// TIA Portal project "项目1_V15.1" (V15.1)

(* hardware
DEVICE "S7-1200 station_2"  S7-1200 Station
   slot 0: "Rack_0"  S7-1200 Rack  Rack  V1.0
   slot 1: "300-1PLC"  CPU 1214C DC/DC/DC  6ES7 214-1AG40-0XB0  V4.2
   slot 2: "DI 16/DQ 16x24VDC_1"  6ES7 223-1BL32-0XB0  V2.0
   slot 3: "DI 16/DQ 16x24VDC_2"  6ES7 223-1BL32-0XB0  V2.0
   slot 4: "DI 8x24VDC_1"  6ES7 221-1BF32-0XB0  V2.0
   slot 5: "AI 4x13BIT/AQ 2x14BIT_1"  6ES7 234-4HE32-0XB0  V2.0
DEVICE "GSD device_9"  GSD.Device.PN
   slot 0: "机架"  Rack  V1.0
   slot 0: "输入轴伺服"  SINAMICS V90 PN V1.0  6SL3 210-5Fxxx-xxFx  V1.00
      slot 0: "SINAMICS V90 PN V1.0"  SINAMICS V90 PN V1.0
      slot 1: "PN-IO"  PN-IO
         slot 1: "端口1"  Port 1
         slot 2: "端口2"  Port 2
      slot 1: "驱动_1"  Drive
         slot 0: "模块访问点"  Module Access Point
         slot 1: "没有 PROFIsafe"  without PROFIsafe
   slot 2: "标准报文3, PZD-5/9"  Standard telegram 3, PZD-5/9
DEVICE "GSD device_8"  GSD.Device.PN
   slot 0: "机架"  Rack  V1.0
   slot 0: "输入轴移载"  SINAMICS V90 PN V1.0  6SL3 210-5Fxxx-xxFx  V1.00
      slot 0: "SINAMICS V90 PN V1.0"  SINAMICS V90 PN V1.0
      slot 1: "PN-IO"  PN-IO
         slot 1: "端口1"  Port 1
         slot 2: "端口2"  Port 2
      slot 1: "驱动_1"  Drive
         slot 0: "模块访问点"  Module Access Point
         slot 1: "没有 PROFIsafe"  without PROFIsafe
   slot 2: "标准报文3, PZD-5/9"  Standard telegram 3, PZD-5/9
DEVICE "GSD device_10"  GSD.Device.PN
   slot 0: "机架"  Rack  V1.0
   slot 0: "工装移载"  SINAMICS V90 PN V1.0  6SL3 210-5Fxxx-xxFx  V1.00
      slot 0: "SINAMICS V90 PN V1.0"  SINAMICS V90 PN V1.0
      slot 1: "PN-IO"  PN-IO
         slot 1: "端口1"  Port 1
         slot 2: "端口2"  Port 2
      slot 1: "驱动_1"  Drive
         slot 0: "模块访问点"  Module Access Point
         slot 1: "没有 PROFIsafe"  without PROFIsafe
   slot 2: "标准报文3, PZD-5/9"  Standard telegram 3, PZD-5/9
*)

// ===== PLC "300-1PLC"  CPU 1214C DC/DC/DC =====

VAR_GLOBAL   // PLC tag table "默认变量表"
   "角度编码器A" AT %I0.0 : Bool;
   "角度编码器B" AT %I0.1 : Bool;
   "角度编码器Z" AT %I0.2 : Bool;
   "在位传感器" AT %I1.4 : Bool;
   "输入轴扶持气缸进到位" AT %I2.0 : Bool;
   "输入轴扶持气缸退到位" AT %I2.1 : Bool;
   "产品夹紧气缸1进到位" AT %I2.2 : Bool;
   "产品夹紧气缸1退到位" AT %I2.3 : Bool;
   "产品夹紧气缸2进到位" AT %I2.5 : Bool;
   "产品夹紧气缸2退到位" AT %I2.4 : Bool;
   "产品定位气缸进到位" AT %I2.6 : Bool;
   "产品定位气缸退到位" AT %I2.7 : Bool;
   "振动检测气缸1进到位" AT %I3.0 : Bool;
   "振动检测气缸1退到位" AT %I3.1 : Bool;
   "振动检测气缸2进到位" AT %I3.2 : Bool;
   "振动检测气缸2退到位" AT %I3.3 : Bool;
   "输出轴花键移载气缸进到位" AT %I3.4 : Bool;
   "输出轴花键移载气缸退到位" AT %I3.5 : Bool;
   "安全门气缸进到位" AT %I3.6 : Bool;
   "安全门气缸退到位" AT %I3.7 : Bool;
   "启动" AT %I4.0 : Bool;
   "复位" AT %I4.1 : Bool;
   "手自动" AT %I4.2 : Bool;
   "安全继电器急停" AT %I4.3 : Bool;
   "安全门开关" AT %I4.4 : Bool;
   "急停" AT %I4.5 : Bool;
   "报警1" AT %I5.0 : Bool;
   "报警2" AT %I5.1 : Bool;
   "报警3" AT %I5.2 : Bool;
   "报警4" AT %I5.3 : Bool;
   "扭矩传感器1" AT %IW144 : Int;
   "扭矩传感器2-1" AT %IW146 : Int;
   "扭矩传感器2-2" AT %IW148 : Int;
   "电流传感器" AT %IW150 : Int;
   "输入轴移载伺服_LowHwLimitSwitch" AT %I0.4 : Bool;
   "输入轴移载伺服_HighHwLimitSwitch" AT %I0.3 : Bool;
   "输入轴移载伺服_归位开关" AT %I0.5 : Bool;
   "工装移载伺服_Drive_IN" AT %I104.0 : "PD_TEL3_IN";
   "工装移载伺服_LowHwLimitSwitch" AT %I0.7 : Bool;
   "工装移载伺服_HighHwLimitSwitch" AT %I0.6 : Bool;
   "工装移载伺服_归位开关" AT %I1.0 : Bool;
   "角度编码器" AT %ID1000 : DInt;
   "气源不足指示" AT %I5.4 : Bool;
   "安全光栅" AT %I4.7 : Bool;
   "工件在位" AT %I1.1 : Bool;
   "输入轴驱动伺服_Drive_IN" AT %I68.0 : "PD_TEL1_IN";
   "输入轴移载伺服_Drive_IN" AT %I86.0 : "PD_TEL3_IN";
   "输入轴驱动伺服_Encoder_IN" AT %I68.0 : "PD_TEL3_IN";
   "复位1" AT %Q0.0 : Bool;
   "复位2" AT %Q0.1 : Bool;
   "复位3" AT %Q0.2 : Bool;
   "复位4" AT %Q0.3 : Bool;
   "点火" AT %Q0.4 : Bool;
   "转速" AT %Q0.5 : Bool;
   "车速" AT %Q0.6 : Bool;
   "输入轴扶持气缸进" AT %Q2.0 : Bool;
   "输入轴扶持气缸退" AT %Q2.1 : Bool;
   "产品松开" AT %Q2.2 : Bool;
   "产品夹紧" AT %Q2.3 : Bool;
   "支架松开" AT %Q2.4 : Bool;
   "支架夹紧" AT %Q2.5 : Bool;
   "产品定位气缸进" AT %Q3.6 : Bool;
   "产品定位气缸退" AT %Q3.7 : Bool;
   "振动检测气缸1进" AT %Q3.0 : Bool;
   "振动检测气缸1退" AT %Q3.1 : Bool;
   "振动检测气缸2进" AT %Q3.2 : Bool;
   "振动检测气缸2退" AT %Q3.3 : Bool;
   "输出轴花键移载气缸进" AT %Q2.6 : Bool;
   "输出轴花键移载气缸退" AT %Q2.7 : Bool;
   "安全门气缸进" AT %Q3.4 : Bool;
   "安全门气缸退" AT %Q3.5 : Bool;
   "三色灯-红" AT %Q4.0 : Bool;
   "三色灯-黄" AT %Q4.1 : Bool;
   "三色灯-绿" AT %Q4.2 : Bool;
   "蜂鸣器" AT %Q4.3 : Bool;
   "两色灯-红" AT %Q4.4 : Bool;
   "两色灯-绿" AT %Q4.5 : Bool;
   "总气阀" AT %Q4.6 : Bool;
   "工位复位中" AT %Q4.7 : Bool;
   "30V电源控制" AT %QW144 : Int;
   "输入轴移载伺服_Drive_OUT" AT %Q74.0 : "PD_TEL3_OUT";
   "工装移载伺服_Drive_OUT" AT %Q84.0 : "PD_TEL3_OUT";
   "输入轴旋转-已复位" AT %Q6.0 : Bool;
   "输入轴移载-已复位" AT %Q6.1 : Bool;
   "工装移载-已复位" AT %Q6.2 : Bool;
   "T1T2切换" AT %Q5.0 : Bool;
   "输入轴驱动伺服_Drive_OUT" AT %Q64.0 : "PD_TEL3_OUT";
   "System_Byte" AT %MB1 : Byte;
   "FirstScan" AT %M1.0 : Bool;
   "DiagStatusUpdate" AT %M1.1 : Bool;
   "AlwaysTRUE" AT %M1.2 : Bool;
   "AlwaysFALSE" AT %M1.3 : Bool;
   "Clock_Byte" AT %MB0 : Byte;
   "Clock_10Hz" AT %M0.0 : Bool;
   "Clock_5Hz" AT %M0.1 : Bool;
   "Clock_2.5Hz" AT %M0.2 : Bool;
   "Clock_2Hz" AT %M0.3 : Bool;
   "Clock_1.25Hz" AT %M0.4 : Bool;
   "Clock_1Hz" AT %M0.5 : Bool;
   "Clock_0.625Hz" AT %M0.6 : Bool;
   "Clock_0.5Hz" AT %M0.7 : Bool;
   "Car_speed" AT %MD2000 : Real;
   "Engine_Speed" AT %MD2004 : Real;
   "复位启动" AT %M100.0 : Bool;
   "复位完成" AT %M100.1 : Bool;
   "程序停止" AT %M100.2 : Bool;
   "电机控制器启动" AT %M99.0 : Bool;
   "电机正转启动" AT %M99.1 : Bool;
   "电机反转启动" AT %M99.2 : Bool;
   "Tag_1" AT %MW1000 : Word;
   "Tag_2" AT %MW1024 : Word;
   "Tag_3" AT %MW1345 : Word;
   "Tag_4" AT %MW1456 : Word;
   "转速方向" AT %Q0.7 : Bool;
   "车速方向" AT %Q1.0 : Bool;
END_VAR

TYPE "In_config"
VERSION : 0.1
   STRUCT
      接近位移 : Real;
      接近速度 : Real;
      套入位移 : Real;
      套入速度 : Real;
      摆动参数 : "In_swing_config";
   END_STRUCT;
END_TYPE

TYPE "In_swing_config"
VERSION : 0.1
   STRUCT
      启用状态 : Real;
      摆动速度 : Real;
      摆动角度 : Real;
      保护扭矩 : Real;
   END_STRUCT;
END_TYPE

TYPE "Fixture_transfer_config"
VERSION : 0.1
   STRUCT
      定位位置 : Real;
      定位速度 : Real;
   END_STRUCT;
END_TYPE

TYPE "Test_No_Load_CFG"
VERSION : 0.1
   STRUCT
      启用助力 : Real := 0.0;
      空载速度 : Real := 0.0;
      空载位移 : Real := 0.0;
      扭矩保护 : Real := 0.0;
   END_STRUCT;
END_TYPE

TYPE "Test_Function_CFG"
VERSION : 0.1
   STRUCT
      试验速度 : Real;
      试验角度 : Real;
      负载扭矩 : Real;
      保护扭矩 : Real;
   END_STRUCT;
END_TYPE

TYPE "Test_Input&Output_Characteristics_CFG"
VERSION : 0.1
   STRUCT
      试验速度 : Real;
      换向扭矩 : Real;
      模拟车速 : Real;
      模拟发动机转速 : Real;
   END_STRUCT;
END_TYPE

TYPE "Test_NVH"
VERSION : 0.1
   STRUCT
      检测点1 : Real;
      检测点2 : Real;
      正向检测时间 : Real;
      逆向检测时间 : Real;
   END_STRUCT;
END_TYPE

DATA_BLOCK "MB_TCON_Rapid"   // DB5
{ S7_Optimized_Access := 'TRUE' }
VERSION : 0.1
   VAR
      MB_SERVER : TCON_IP_v4;
   END_VAR
BEGIN
   MB_SERVER.InterfaceId := 64;
   MB_SERVER.ID := 1;
   MB_SERVER.LocalPort := 502;
END_DATA_BLOCK

DATA_BLOCK "Modbus_Data_Rapid"   // DB6
{ S7_Optimized_Access := 'FALSE' }
VERSION : 0.1
   VAR
      设备编号 : Int := 0;
      产品型号 : Int := 0;
      设备状态 : Int;
      错误代码 : Int;
      当前曲线 : Int;
      传感器标定值 : Array[0..7] of Real;
   END_VAR
BEGIN
   // 传感器标定值[0] : 输入轴驱动伺服位移
   // 传感器标定值[1] : 输入轴移载伺服位移
   // 传感器标定值[2] : 工装移载伺服位移
   // 传感器标定值[3] : 输入轴编码器
   // 传感器标定值[4] : 输入轴扭矩
   // 传感器标定值[5] : 输出轴扭矩小量程
   // 传感器标定值[6] : 输出轴扭矩大量程
   // 传感器标定值[7] : 吸收电流
END_DATA_BLOCK

DATA_BLOCK "Modbus_Data"   // DB7
{ S7_Optimized_Access := 'FALSE' }
VERSION : 0.1
   VAR
      输入扭矩传感器参数 : Array[0..1] of Real;   // AF400001L2
      输出扭矩传感器参数小量程 : Array[0..1] of Real;   // AF400005L2
      输出扭矩传感器参数大量程 : Array[0..1] of Real;   // AF400009L2
      电流传感器参数 : Array[0..1] of Real;   // AF400013L2
      输入轴自动参数 : "In_config";   // AF400017L4
      输入轴移载手动参数 : Array[0..3] of Real;   // AF400025L4
      输入轴旋转参数 : Array[0..3] of Real;   // AF400041L4
      工装移载参数 : "Fixture_transfer_config";   // AF400049L4
      工装移载手动参数 : Array[0..3] of Real;   // AF400057L4
      空载试验参数 : "Test_No_Load_CFG";   // AF400065L4
      功能试验参数 : "Test_Function_CFG";   // AF400073L4
      力特性试验参数 : "Test_Input&Output_Characteristics_CFG";   // AF400081L4
      逆向空载试验参数 : "Test_No_Load_CFG";   // AF400097L4
      振动NVH试验参数 : "Test_NVH";   // AF400097L4
   END_VAR
BEGIN
   输出扭矩传感器参数小量程[0] := 0.0;   // 量程下限
   输出扭矩传感器参数小量程[1] := 20.0;   // 量程上限
   输出扭矩传感器参数大量程[1] := 233.0;   // 量程上限（校验值233）
   输出扭矩传感器参数大量程[0] := 0.0;   // 量程下限
   输入扭矩传感器参数[1] := 58.0;   // 量程上限(校验值48.0)
   输入扭矩传感器参数[0] := 0.0;   // 量程下限
   电流传感器参数[0] := -100.0;   // 量程下限
   电流传感器参数[1] := 100.0;   // 量程下限
   // 输入轴移载手动参数[0] : 手动状态
   // 输入轴移载手动参数[1] : 手动速度
   // 输入轴移载手动参数[2] : 相对定位
   // 输入轴移载手动参数[3] : 绝对定位
   // 输入轴旋转参数[0] : 手动状态
   // 输入轴旋转参数[1] : 手动速度
   // 输入轴旋转参数[2] : 相对定位
   // 输入轴旋转参数[3] : 绝对定位
   // 工装移载手动参数[0] : 手动状态
   // 工装移载手动参数[1] : 手动速度
   // 工装移载手动参数[2] : 相对定位
   // 工装移载手动参数[3] : 绝对定位
END_DATA_BLOCK

DATA_BLOCK "MB_TCON"   // DB9
{ S7_Optimized_Access := 'TRUE' }
VERSION : 0.1
   VAR
      MB_SERVER : TCON_IP_v4;
   END_VAR
BEGIN
   MB_SERVER.InterfaceId := 64;
   MB_SERVER.ID := 2;
   MB_SERVER.LocalPort := 502;
END_DATA_BLOCK

DATA_BLOCK "Reset_DB"   // DB11
{ S7_Optimized_Access := 'TRUE' }
VERSION : 0.1
// stored: InstanceOfName Reset
"Reset"
BEGIN
END_DATA_BLOCK

DATA_BLOCK "Alarm_DB"   // DB15
{ S7_Optimized_Access := 'TRUE' }
VERSION : 0.1
// stored: InstanceOfName Alarm
"Alarm"
BEGIN
END_DATA_BLOCK

DATA_BLOCK "All_Servo_DB"   // DB18
{ S7_Optimized_Access := 'TRUE' }
VERSION : 0.1
// stored: InstanceOfName All_Servo
"All_Servo"
BEGIN
END_DATA_BLOCK

DATA_BLOCK "设置电压_DB"   // DB20
{ S7_Optimized_Access := 'TRUE' }
VERSION : 0.1
// stored: InstanceOfName 设置电压
"设置电压"
BEGIN
END_DATA_BLOCK

DATA_BLOCK "Auto_DB"   // DB21
{ S7_Optimized_Access := 'TRUE' }
VERSION : 0.1
// stored: InstanceOfName Auto
"Auto"
BEGIN
END_DATA_BLOCK

DATA_BLOCK "左右摆动_DB"   // DB22
{ S7_Optimized_Access := 'TRUE' }
VERSION : 0.1
// stored: InstanceOfName 左右摆动
"左右摆动"
BEGIN
END_DATA_BLOCK

// folder: System blocks/Program resources

DATA_BLOCK "IEC_Timer_0_DB"   // DB19
{ S7_Optimized_Access := 'TRUE' }
AUTHOR : Simatic
FAMILY : IEC
NAME : IEC_TMR
VERSION : 1.0
// stored: InstanceOfName IEC_TIMER
"IEC_TIMER"
BEGIN
END_DATA_BLOCK

// folder: (top level)

DATA_BLOCK "输入轴驱动伺服"   // DB1, Motion_DB
{ S7_Optimized_Access := 'TRUE' }
AUTHOR : SIMATIC
FAMILY : BasicMC
NAME : TO_PosAx
VERSION : 6.0
// stored: InstanceOfName TO_PositioningAxis
"TO_PositioningAxis"
BEGIN
   // Axis.Encoder.TelegramAddressOutCU = %Q64.0
   // Axis.Encoder.TelegramAddressInCU = %I68.0
   // Axis.Encoder.DoNameCU = 输入轴伺服.驱动_1_编码器1
   // Axis.Drive.OutputAddress = 64
   // Axis.Drive.InputAddress = 68
   // Axis.Encoder.OutputAddress = 64
   // Axis.Encoder.InputAddress = 68
   // Axis.Drive.TelegramAddressOutCU = %Q64.0
   // Axis.Drive.TelegramAddressInCU = %I68.0
   // Axis.Drive.TelegramType = 2
   // Axis.Drive.DoNameCU = 输入轴伺服.驱动_1
   // Axis.LengthUnit.LastDistance = 1005
   // Axis.LengthUnitNormalized.Distance = 1005
   // Axis.Encoder.SelectedHscIndexCU = -1
   // Axis.Encoder.DbTypeCU = Classic
   // Axis.Drive.DbTypeCU = Classic
END_DATA_BLOCK

DATA_BLOCK "输入轴移载伺服"   // DB2, Motion_DB
{ S7_Optimized_Access := 'TRUE' }
AUTHOR : SIMATIC
FAMILY : BasicMC
NAME : TO_PosAx
VERSION : 6.0
// stored: InstanceOfName TO_PositioningAxis
"TO_PositioningAxis"
BEGIN
   // Axis.Encoder.TelegramAddressOutCU = %Q74.0
   // Axis.Encoder.TelegramAddressInCU = %I86.0
   // Axis.Encoder.DoNameCU = 输入轴移载.驱动_1_编码器1
   // Axis.Drive.OutputAddress = 74
   // Axis.Drive.InputAddress = 86
   // Axis.Encoder.OutputAddress = 74
   // Axis.Encoder.InputAddress = 86
   // Axis.Drive.TelegramAddressOutCU = %Q74.0
   // Axis.Drive.TelegramAddressInCU = %I86.0
   // Axis.Drive.TelegramType = 2
   // Axis.Drive.DoNameCU = 输入轴移载.驱动_1
   // Axis.HomingReferencePointSwitch_AddressCU = %I0.5
   // Axis.PositionLimitsMax_AddressCU = %I0.3
   // Axis.PositionLimitsMin_AddressCU = %I0.4
   // Axis.LengthUnitNormalized.Distance = 1013
   // Axis.Encoder.SelectedHscIndexCU = -1
   // Axis.Encoder.DbTypeCU = Classic
   // Axis.Drive.DbTypeCU = Classic
END_DATA_BLOCK

DATA_BLOCK "工装移载伺服"   // DB3, Motion_DB
{ S7_Optimized_Access := 'TRUE' }
AUTHOR : SIMATIC
FAMILY : BasicMC
NAME : TO_PosAx
VERSION : 6.0
// stored: InstanceOfName TO_PositioningAxis
"TO_PositioningAxis"
BEGIN
   // Axis.Encoder.TelegramAddressOutCU = %Q84.0
   // Axis.Encoder.TelegramAddressInCU = %I104.0
   // Axis.Encoder.DoNameCU = 工装移载.驱动_1_编码器1
   // Axis.Drive.OutputAddress = 84
   // Axis.Drive.InputAddress = 104
   // Axis.Encoder.OutputAddress = 84
   // Axis.Encoder.InputAddress = 104
   // Axis.Drive.TelegramAddressOutCU = %Q84.0
   // Axis.Drive.TelegramAddressInCU = %I104.0
   // Axis.Drive.DoNameCU = 工装移载.驱动_1
   // Axis.HomingReferencePointSwitch_AddressCU = %I1.0
   // Axis.PositionLimitsMax_AddressCU = %I0.6
   // Axis.PositionLimitsMin_AddressCU = %I0.7
   // Axis.Drive.TelegramType = 2
   // Axis.LengthUnitNormalized.Distance = 1013
   // Axis.Encoder.SelectedHscIndexCU = -1
   // Axis.Encoder.DbTypeCU = Classic
   // Axis.Drive.DbTypeCU = Classic
END_DATA_BLOCK

DATA_BLOCK "模拟转速"   // DB16, Motion_DB
{ S7_Optimized_Access := 'TRUE' }
AUTHOR : SIMATIC
FAMILY : BasicMC
NAME : TO_PosAx
VERSION : 6.0
// stored: InstanceOfName TO_PositioningAxis
"TO_PositioningAxis"
BEGIN
   // Axis.OnlinePtoIndexCU = 3
   // Axis.SelectedChannel2EnumCU = %Q1.0
   // Axis.LengthUnit.LastDistance = -1
   // Axis.OnlinePtoModeCUEnumValue = PTO（脉冲 A 和方向 B）
   // Axis.OnlinePtoModeCU = 16#0000_0002
   // Axis.SelectedChannel1EnumCU = %Q0.5
   // Pulse.MinDeltaDeltaFrequencyCU = 0.004
   // Pulse.MaxDeltaDeltaFrequencyCU = 1.0E+10
   // Pulse.MinDeltaFrequencyCU = 0.005
   // Pulse.MaxDeltaFrequencyCU = 9.5E+9
   // Pulse.MinFrequencyCU = 1.0
   // Pulse.MaxFrequencyCU = 30000.0
   // Pulse.OutputSourceCU = 16#0000_0000
   // Axis.SelectPTO = 3
END_DATA_BLOCK

DATA_BLOCK "模拟车速"   // DB17, Motion_DB
{ S7_Optimized_Access := 'TRUE' }
AUTHOR : SIMATIC
FAMILY : BasicMC
NAME : TO_PosAx
VERSION : 6.0
// stored: InstanceOfName TO_PositioningAxis
"TO_PositioningAxis"
BEGIN
   // Axis.OnlinePtoIndexCU = 2
   // Axis.OnlinePtoModeCU = 16#0000_0002
   // Axis.SelectedChannel2EnumCU = %Q0.7
   // Axis.SelectedChannel1EnumCU = %Q0.6
   // Pulse.MinDeltaDeltaFrequencyCU = 0.004
   // Pulse.MaxDeltaDeltaFrequencyCU = 1.0E+10
   // Pulse.MinDeltaFrequencyCU = 0.005
   // Pulse.MaxDeltaFrequencyCU = 9.5E+9
   // Pulse.MinFrequencyCU = 1.0
   // Pulse.MaxFrequencyCU = 30000.0
   // Pulse.OutputSourceCU = 16#0000_0000
   // Axis.SelectPTO = 2
   // Axis.OnlinePtoModeCUEnumValue = PTO（脉冲 A 和方向 B）
   // Axis.LengthUnit.LastDistance = -1
END_DATA_BLOCK

FUNCTION_BLOCK "设置电压"   // FB1, LAD
{ S7_Optimized_Access := 'TRUE' }
VERSION : 0.1
   VAR_INPUT
      电压 : Real;
   END_VAR
BEGIN

REGION Network 1
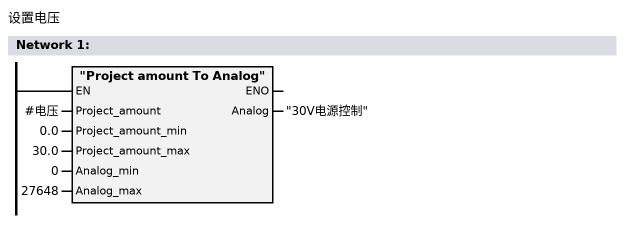
   RUNG wire#powerrail
      "Project amount To Analog"(Project_amount := #电压, Project_amount_min := 0.0, Project_amount_max := 30.0, Analog_min := 0, Analog_max := 27648, Analog => "30V电源控制")
   END_RUNG
   // the same network as SCL:
   "Project amount To Analog"(Project_amount := #电压,
                           Project_amount_min := 0.0,
                           Project_amount_max := 30.0,
                           Analog_min := 0,
                           Analog_max := 27648,
                           Analog => "30V电源控制");
END_REGION
END_FUNCTION_BLOCK

FUNCTION_BLOCK "Servo"   // FB2, LAD
{ S7_Optimized_Access := 'TRUE' }
VERSION : 0.1
   VAR_INPUT
      Axis : TO_PositioningAxis;
      Son : Bool;
      Halt : Bool;
      Stop : Bool;
      Absoulte_Position : Real;
      Relative_Position : Real;
      Velocity : Real;
      JogForword : Bool;
      JogBackword : Bool;
      MoveAbsolute : Bool;
      MoveRelative : Bool;
      MoveHome : Bool;
      Mode : Int;
   END_VAR
   VAR_OUTPUT
      Done : Bool;
   END_VAR
   VAR_IN_OUT
      HomingDone : Bool;
   END_VAR
   VAR
      Temp : Array[0..7] of Bool;
      Reser_Done : Bool;
      MC_Power_Instance : MC_Power;
      MC_Reset_Instance : MC_Reset;
      MC_Home_Instance : MC_Home;
      MC_Halt_Instance : MC_Halt;
      MC_MoveAbsolute_Instance : MC_MoveAbsolute;
      MC_MoveRelative_Instance : MC_MoveRelative;
      MC_MoveJog_Instance : MC_MoveJog;
      IEC_Timer_0_Instance : TP_TIME;
      IEC_Timer_0_Instance_1 : TON_TIME;
      IEC_Timer_0_Instance_2 : TON_TIME;
      MC_ReadParam_Instance : MC_ReadParam;
   END_VAR
   VAR_TEMP   // added for the SCL form of the ladder/FBD networks
      _w1 : Bool;
   END_VAR
BEGIN

REGION Network 1
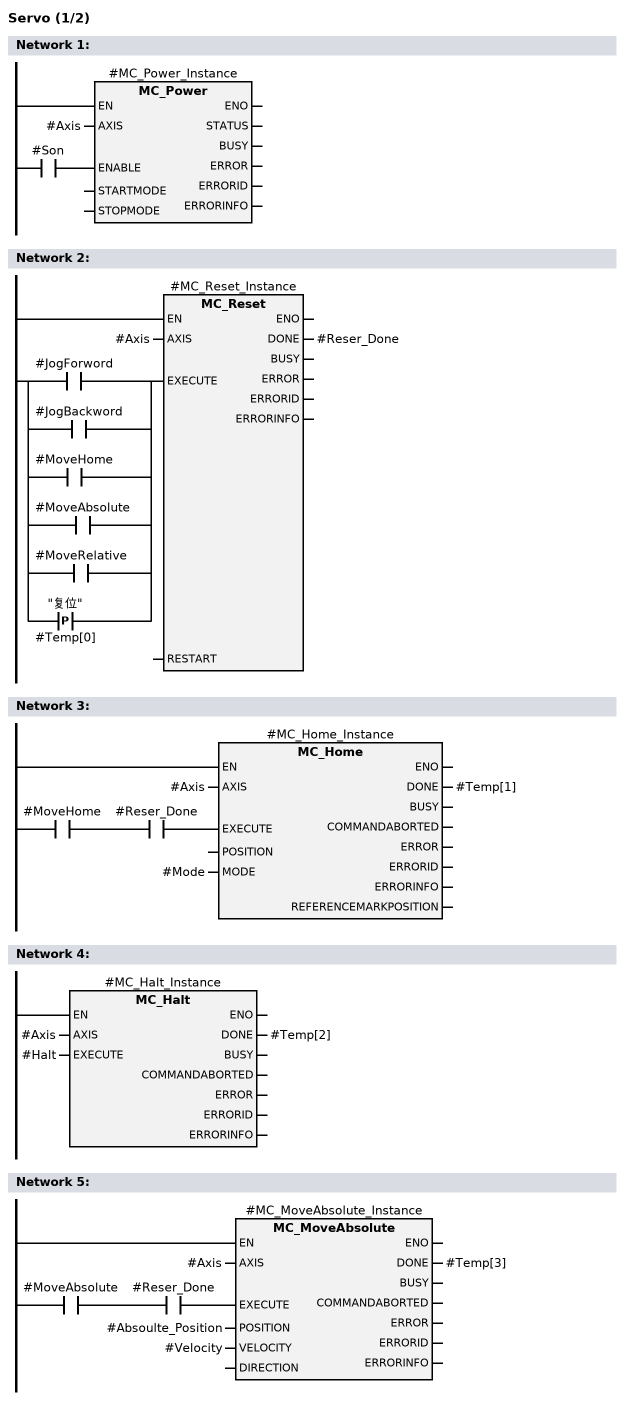
   #MC_Power_Instance(Axis := #Axis, Enable := #Son);   // MC_Power
END_REGION

REGION Network 2
   #_w1 := "复位" AND NOT #Temp[0];   // rising edge of "复位"
   #Temp[0] := "复位";
   #MC_Reset_Instance(Axis := #Axis,   // MC_Reset
                      Execute := #JogForword OR #JogBackword OR #MoveHome OR #MoveAbsolute OR #MoveRelative OR #_w1,
                      Done => #Reser_Done);
END_REGION

REGION Network 3
   #MC_Home_Instance(Axis := #Axis, Execute := #MoveHome AND #Reser_Done, Mode := #Mode, Done => #Temp[1]);   // MC_Home
END_REGION

REGION Network 4
   #MC_Halt_Instance(Axis := #Axis, Execute := #Halt, Done => #Temp[2]);   // MC_Halt
END_REGION

REGION Network 5
   #MC_MoveAbsolute_Instance(Axis := #Axis,   // MC_MoveAbsolute
                           Execute := #MoveAbsolute AND #Reser_Done,
                           Position := #Absoulte_Position,
                           Velocity := #Velocity,
                           Done => #Temp[3]);
END_REGION

REGION Network 6
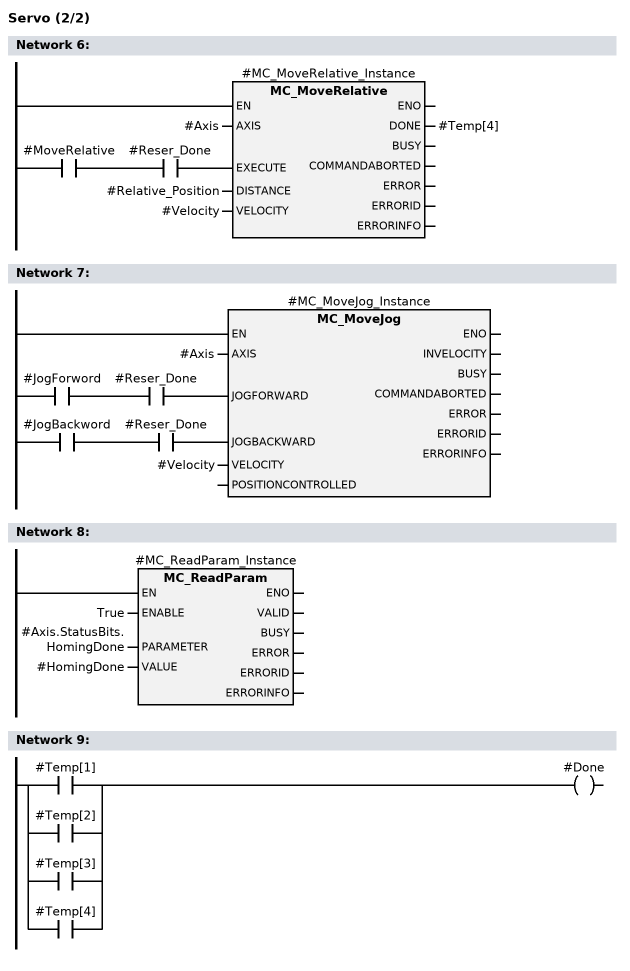
   #MC_MoveRelative_Instance(Axis := #Axis,   // MC_MoveRelative
                           Execute := #MoveRelative AND #Reser_Done,
                           Distance := #Relative_Position,
                           Velocity := #Velocity,
                           Done => #Temp[4]);
END_REGION

REGION Network 7
   #MC_MoveJog_Instance(Axis := #Axis,   // MC_MoveJog
                        JogForward := #JogForword AND #Reser_Done,
                        JogBackward := #JogBackword AND #Reser_Done,
                        Velocity := #Velocity);
END_REGION

REGION Network 8
   #MC_ReadParam_Instance(Enable := True, Parameter := #Axis.StatusBits.HomingDone, Value := #HomingDone);   // MC_ReadParam
END_REGION

REGION Network 9
   RUNG wire#powerrail
      Contact( #Temp[1] )
      wire#w1
      Coil( #Done )
   END_RUNG
   RUNG wire#powerrail
      Contact( #Temp[2] )
   END_RUNG wire#w1
   RUNG wire#powerrail
      Contact( #Temp[3] )
   END_RUNG wire#w1
   RUNG wire#powerrail
      Contact( #Temp[4] )
   END_RUNG wire#w1
   // the same network as SCL:
   #Done := #Temp[1] OR #Temp[2] OR #Temp[3] OR #Temp[4];
END_REGION
END_FUNCTION_BLOCK

FUNCTION_BLOCK "All_Servo"   // FB3, LAD
{ S7_Optimized_Access := 'TRUE' }
VERSION : 0.1
   VAR
      Temp : Array[0..3] of Bool;
      IEC_Timer_0_Instance : TON_TIME;
      IEC_Timer_0_Instance_1 : TP_TIME;
      IEC_Timer_0_Instance_2 : TP_TIME;
      IEC_Timer_0_Instance_3 : TON_TIME;
      IEC_Timer_0_Instance_4 : TP_TIME;
      IEC_Timer_0_Instance_5 : TON_TIME;
      IEC_Timer_0_Instance_6 : TON_TIME;
      Servo_Instance : "Servo";
      Servo_Instance_1 : "Servo";
      Servo_Instance_2 : "Servo";
      Servo_Instance_3 : "Servo";
      MC_Power_Instance : MC_Power;
      MC_Power_Instance_1 : MC_Power;
   END_VAR
   VAR_TEMP   // added for the SCL form of the ladder/FBD networks
      _w1 : Bool;
   END_VAR
BEGIN

REGION Network 1: 输入轴驱动伺服
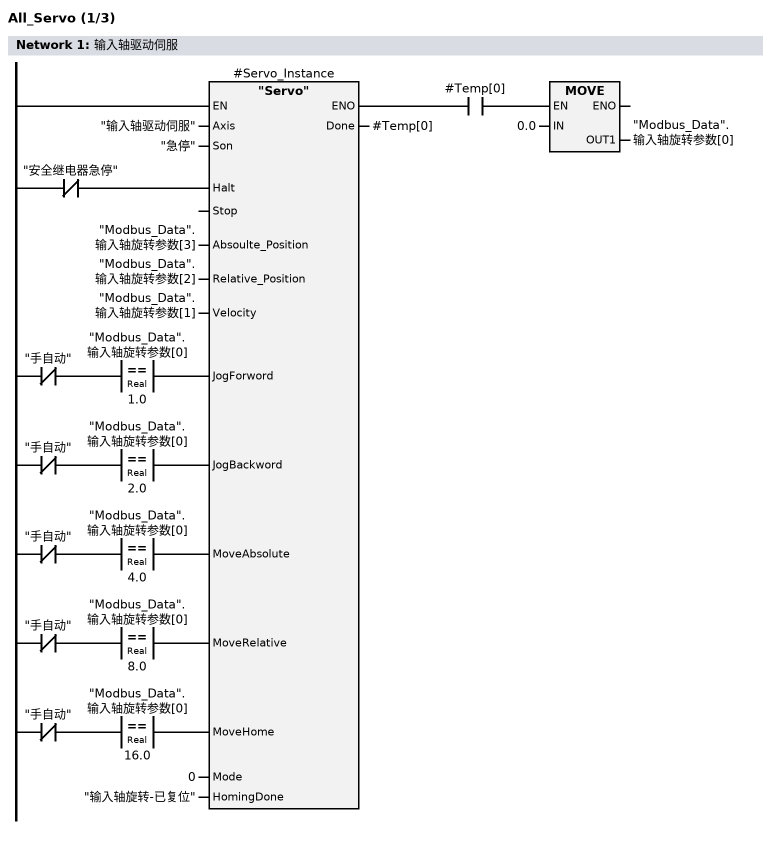
   RUNG wire#powerrail
      #Servo_Instance(Halt := wire#w1, JogForword := wire#w2, JogBackword := wire#w3, MoveAbsolute := wire#w4, MoveRelative := wire#w5, MoveHome := wire#w6, Axis := "输入轴驱动伺服", Son := "急停", Stop :=, Absoulte_Position := "Modbus_Data".输入轴旋转参数[3], Relative_Position := "Modbus_Data".输入轴旋转参数[2], Velocity := "Modbus_Data".输入轴旋转参数[1], Mode := 0, HomingDone := "输入轴旋转-已复位", Done => #Temp[0])
      Contact( #Temp[0] )
      Move(in := 0.0, out1 => "Modbus_Data".输入轴旋转参数[0])
   END_RUNG
   RUNG wire#powerrail
      I_Contact( "安全继电器急停" )
   END_RUNG wire#w1
   RUNG wire#powerrail
      I_Contact( "手自动" )
      { S7_Templates := "SrcType := Real" } EQ_Contact(in1 := "Modbus_Data".输入轴旋转参数[0], in2 := 1.0)
   END_RUNG wire#w2
   RUNG wire#powerrail
      I_Contact( "手自动" )
      { S7_Templates := "SrcType := Real" } EQ_Contact(in1 := "Modbus_Data".输入轴旋转参数[0], in2 := 2.0)
   END_RUNG wire#w3
   RUNG wire#powerrail
      I_Contact( "手自动" )
      { S7_Templates := "SrcType := Real" } EQ_Contact(in1 := "Modbus_Data".输入轴旋转参数[0], in2 := 4.0)
   END_RUNG wire#w4
   RUNG wire#powerrail
      I_Contact( "手自动" )
      { S7_Templates := "SrcType := Real" } EQ_Contact(in1 := "Modbus_Data".输入轴旋转参数[0], in2 := 8.0)
   END_RUNG wire#w5
   RUNG wire#powerrail
      I_Contact( "手自动" )
      { S7_Templates := "SrcType := Real" } EQ_Contact(in1 := "Modbus_Data".输入轴旋转参数[0], in2 := 16.0)
   END_RUNG wire#w6
   // the same network as SCL:
   #Servo_Instance(Axis := "输入轴驱动伺服",   // "Servo"
                   Son := "急停",
                   Halt := NOT "安全继电器急停",
                   Absoulte_Position := "Modbus_Data".输入轴旋转参数[3],
                   Relative_Position := "Modbus_Data".输入轴旋转参数[2],
                   Velocity := "Modbus_Data".输入轴旋转参数[1],
                   JogForword := NOT "手自动" AND ("Modbus_Data".输入轴旋转参数[0] = 1.0),
                   JogBackword := NOT "手自动" AND ("Modbus_Data".输入轴旋转参数[0] = 2.0),
                   MoveAbsolute := NOT "手自动" AND ("Modbus_Data".输入轴旋转参数[0] = 4.0),
                   MoveRelative := NOT "手自动" AND ("Modbus_Data".输入轴旋转参数[0] = 8.0),
                   MoveHome := NOT "手自动" AND ("Modbus_Data".输入轴旋转参数[0] = 16.0),
                   Mode := 0,
                   HomingDone := "输入轴旋转-已复位",
                   Done => #Temp[0],
                   ENO => #_w1);
   IF #_w1 AND #Temp[0] THEN "Modbus_Data".输入轴旋转参数[0] := 0.0; END_IF;
END_REGION

REGION Network 2: 输入轴移载伺服
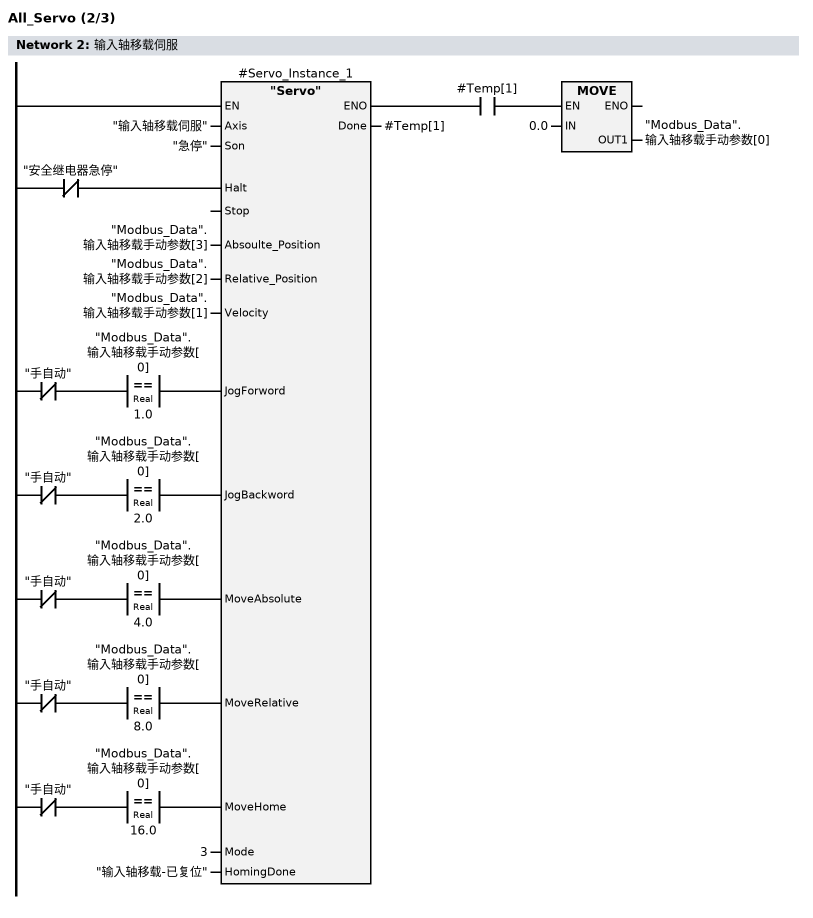
   RUNG wire#powerrail
      #Servo_Instance_1(Halt := wire#w1, JogForword := wire#w2, JogBackword := wire#w3, MoveAbsolute := wire#w4, MoveRelative := wire#w5, MoveHome := wire#w6, Axis := "输入轴移载伺服", Son := "急停", Stop :=, Absoulte_Position := "Modbus_Data".输入轴移载手动参数[3], Relative_Position := "Modbus_Data".输入轴移载手动参数[2], Velocity := "Modbus_Data".输入轴移载手动参数[1], Mode := 3, HomingDone := "输入轴移载-已复位", Done => #Temp[1])
      Contact( #Temp[1] )
      Move(in := 0.0, out1 => "Modbus_Data".输入轴移载手动参数[0])
   END_RUNG
   RUNG wire#powerrail
      I_Contact( "安全继电器急停" )
   END_RUNG wire#w1
   RUNG wire#powerrail
      I_Contact( "手自动" )
      { S7_Templates := "SrcType := Real" } EQ_Contact(in1 := "Modbus_Data".输入轴移载手动参数[0], in2 := 1.0)
   END_RUNG wire#w2
   RUNG wire#powerrail
      I_Contact( "手自动" )
      { S7_Templates := "SrcType := Real" } EQ_Contact(in1 := "Modbus_Data".输入轴移载手动参数[0], in2 := 2.0)
   END_RUNG wire#w3
   RUNG wire#powerrail
      I_Contact( "手自动" )
      { S7_Templates := "SrcType := Real" } EQ_Contact(in1 := "Modbus_Data".输入轴移载手动参数[0], in2 := 4.0)
   END_RUNG wire#w4
   RUNG wire#powerrail
      I_Contact( "手自动" )
      { S7_Templates := "SrcType := Real" } EQ_Contact(in1 := "Modbus_Data".输入轴移载手动参数[0], in2 := 8.0)
   END_RUNG wire#w5
   RUNG wire#powerrail
      I_Contact( "手自动" )
      { S7_Templates := "SrcType := Real" } EQ_Contact(in1 := "Modbus_Data".输入轴移载手动参数[0], in2 := 16.0)
   END_RUNG wire#w6
   // the same network as SCL:
   #Servo_Instance_1(Axis := "输入轴移载伺服",   // "Servo"
                     Son := "急停",
                     Halt := NOT "安全继电器急停",
                     Absoulte_Position := "Modbus_Data".输入轴移载手动参数[3],
                     Relative_Position := "Modbus_Data".输入轴移载手动参数[2],
                     Velocity := "Modbus_Data".输入轴移载手动参数[1],
                     JogForword := NOT "手自动" AND ("Modbus_Data".输入轴移载手动参数[0] = 1.0),
                     JogBackword := NOT "手自动" AND ("Modbus_Data".输入轴移载手动参数[0] = 2.0),
                     MoveAbsolute := NOT "手自动" AND ("Modbus_Data".输入轴移载手动参数[0] = 4.0),
                     MoveRelative := NOT "手自动" AND ("Modbus_Data".输入轴移载手动参数[0] = 8.0),
                     MoveHome := NOT "手自动" AND ("Modbus_Data".输入轴移载手动参数[0] = 16.0),
                     Mode := 3,
                     HomingDone := "输入轴移载-已复位",
                     Done => #Temp[1],
                     ENO => #_w1);
   IF #_w1 AND #Temp[1] THEN "Modbus_Data".输入轴移载手动参数[0] := 0.0; END_IF;
END_REGION

REGION Network 3: 工装移载伺服
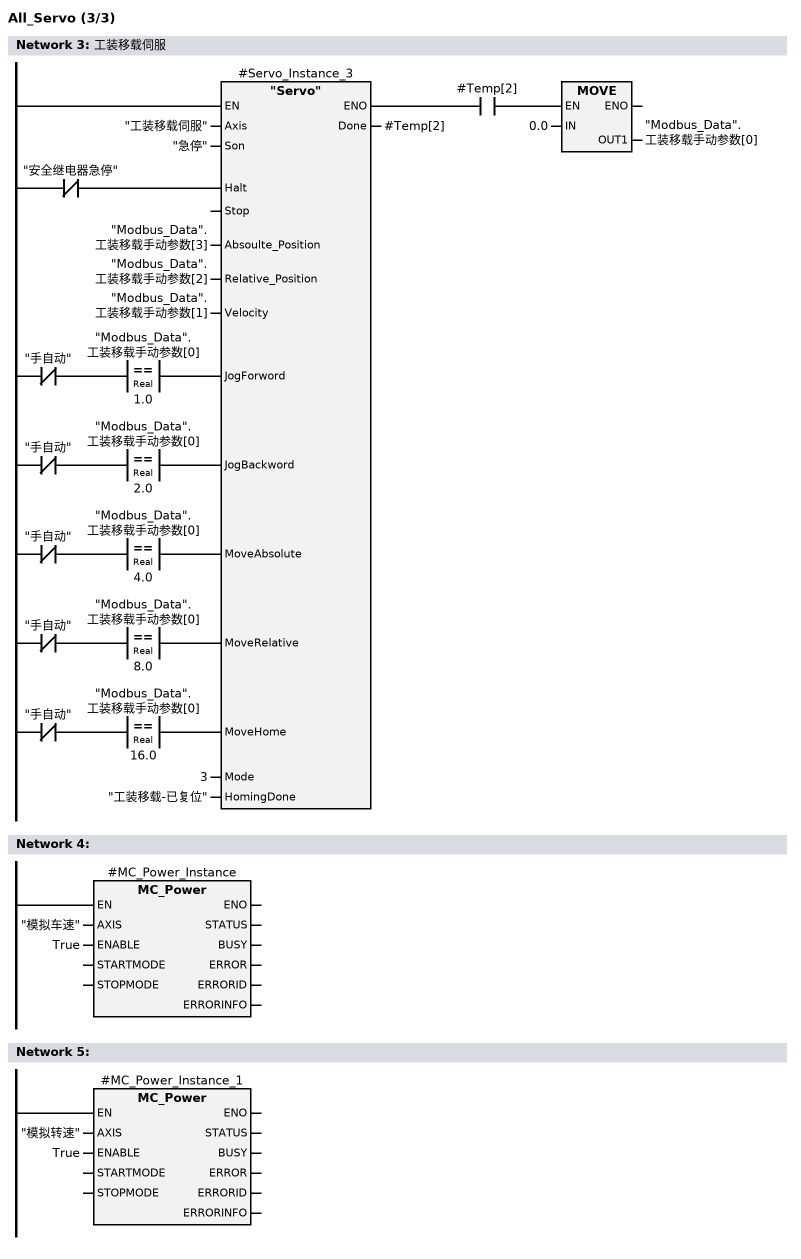
   RUNG wire#powerrail
      #Servo_Instance_3(Halt := wire#w1, JogForword := wire#w2, JogBackword := wire#w3, MoveAbsolute := wire#w4, MoveRelative := wire#w5, MoveHome := wire#w6, Axis := "工装移载伺服", Son := "急停", Stop :=, Absoulte_Position := "Modbus_Data".工装移载手动参数[3], Relative_Position := "Modbus_Data".工装移载手动参数[2], Velocity := "Modbus_Data".工装移载手动参数[1], Mode := 3, HomingDone := "工装移载-已复位", Done => #Temp[2])
      Contact( #Temp[2] )
      Move(in := 0.0, out1 => "Modbus_Data".工装移载手动参数[0])
   END_RUNG
   RUNG wire#powerrail
      I_Contact( "安全继电器急停" )
   END_RUNG wire#w1
   RUNG wire#powerrail
      I_Contact( "手自动" )
      { S7_Templates := "SrcType := Real" } EQ_Contact(in1 := "Modbus_Data".工装移载手动参数[0], in2 := 1.0)
   END_RUNG wire#w2
   RUNG wire#powerrail
      I_Contact( "手自动" )
      { S7_Templates := "SrcType := Real" } EQ_Contact(in1 := "Modbus_Data".工装移载手动参数[0], in2 := 2.0)
   END_RUNG wire#w3
   RUNG wire#powerrail
      I_Contact( "手自动" )
      { S7_Templates := "SrcType := Real" } EQ_Contact(in1 := "Modbus_Data".工装移载手动参数[0], in2 := 4.0)
   END_RUNG wire#w4
   RUNG wire#powerrail
      I_Contact( "手自动" )
      { S7_Templates := "SrcType := Real" } EQ_Contact(in1 := "Modbus_Data".工装移载手动参数[0], in2 := 8.0)
   END_RUNG wire#w5
   RUNG wire#powerrail
      I_Contact( "手自动" )
      { S7_Templates := "SrcType := Real" } EQ_Contact(in1 := "Modbus_Data".工装移载手动参数[0], in2 := 16.0)
   END_RUNG wire#w6
   // the same network as SCL:
   #Servo_Instance_3(Axis := "工装移载伺服",   // "Servo"
                     Son := "急停",
                     Halt := NOT "安全继电器急停",
                     Absoulte_Position := "Modbus_Data".工装移载手动参数[3],
                     Relative_Position := "Modbus_Data".工装移载手动参数[2],
                     Velocity := "Modbus_Data".工装移载手动参数[1],
                     JogForword := NOT "手自动" AND ("Modbus_Data".工装移载手动参数[0] = 1.0),
                     JogBackword := NOT "手自动" AND ("Modbus_Data".工装移载手动参数[0] = 2.0),
                     MoveAbsolute := NOT "手自动" AND ("Modbus_Data".工装移载手动参数[0] = 4.0),
                     MoveRelative := NOT "手自动" AND ("Modbus_Data".工装移载手动参数[0] = 8.0),
                     MoveHome := NOT "手自动" AND ("Modbus_Data".工装移载手动参数[0] = 16.0),
                     Mode := 3,
                     HomingDone := "工装移载-已复位",
                     Done => #Temp[2],
                     ENO => #_w1);
   IF #_w1 AND #Temp[2] THEN "Modbus_Data".工装移载手动参数[0] := 0.0; END_IF;
END_REGION

REGION Network 4
   #MC_Power_Instance(Axis := "模拟车速", Enable := True);   // MC_Power
END_REGION

REGION Network 5
   #MC_Power_Instance_1(Axis := "模拟转速", Enable := True);   // MC_Power
END_REGION
END_FUNCTION_BLOCK

FUNCTION_BLOCK "Reset"   // FB4, LAD
{ S7_Optimized_Access := 'TRUE' }
VERSION : 0.1
   VAR_INPUT
      Start : Bool;
      Stop : Bool;
   END_VAR
   VAR_OUTPUT
      Done : Bool;
   END_VAR
   VAR
      P1 : Real;
      P2 : Real;
      "Step" : Int;
      Temp : Array[0..10] of Bool;
      MC_Home_Instance : MC_Home;
      MC_Home_Instance_1 : MC_Home;
      CTRL_HSC_0_Instance : CTRL_HSC;
      MC_Home_Instance_2 : MC_Home;
      MC_MoveAbsolute_Instance : MC_MoveAbsolute;
      IEC_Timer_0_Instance : TON_TIME;
   END_VAR
   VAR_TEMP   // added for the SCL form of the ladder/FBD networks
      _w1 : Bool;
      _w2 : Bool;
      _w3 : Bool;
   END_VAR
BEGIN

REGION Network 1
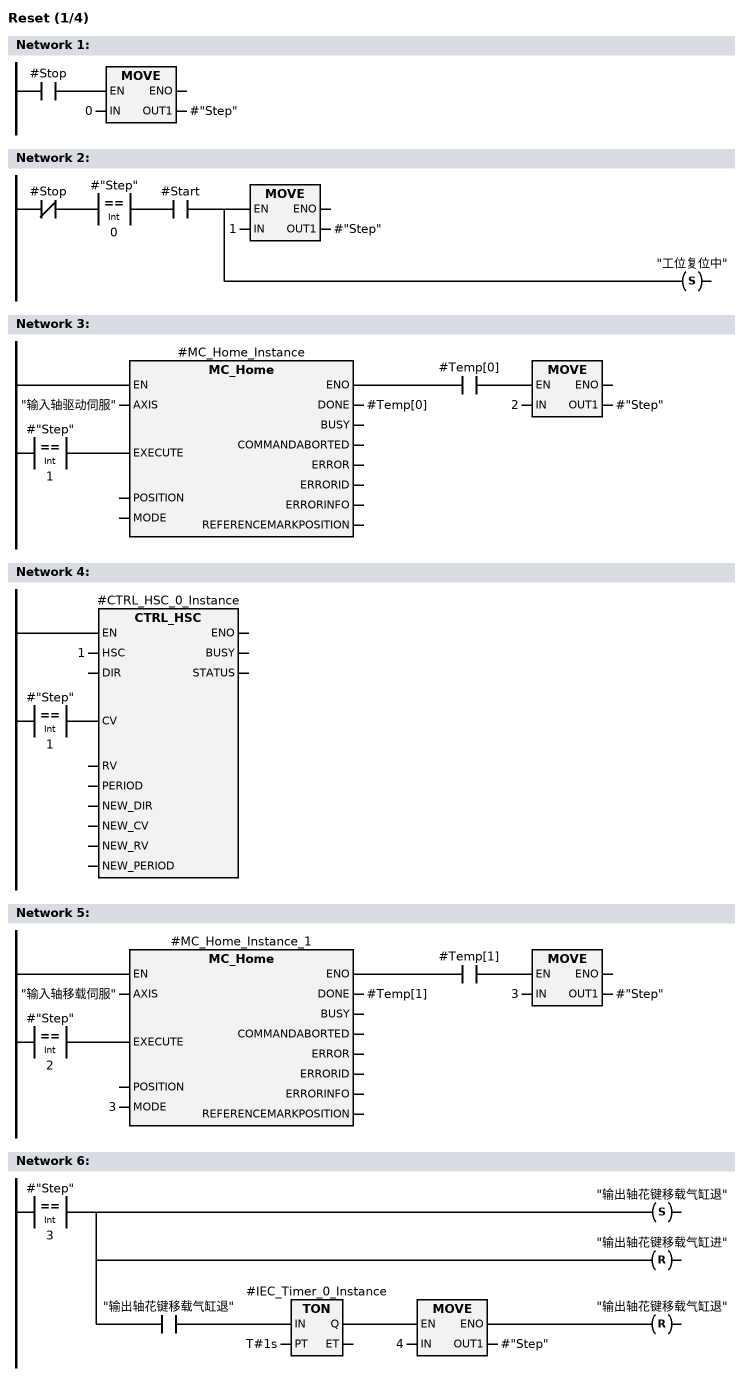
   RUNG wire#powerrail
      Contact( #Stop )
      Move(in := 0, out1 => #"Step")
   END_RUNG
   // the same network as SCL:
   IF #Stop THEN #"Step" := 0; END_IF;
END_REGION

REGION Network 2
   RUNG wire#powerrail
      I_Contact( #Stop )
      { S7_Templates := "SrcType := Int" } EQ_Contact(in1 := #"Step", in2 := 0)
      Contact( #Start )
      wire#w1
      Move(in := 1, out1 => #"Step")
   END_RUNG
   RUNG wire#w1
      S_Coil( "工位复位中" )
   END_RUNG
   // the same network as SCL:
   #_w1 := NOT #Stop AND (#"Step" = 0) AND #Start;
   IF #_w1 THEN
       #"Step" := 1;
       "工位复位中" := TRUE;
   END_IF;
END_REGION

REGION Network 3
   // ENO of a box is taken as its EN; it also drops when the box reports an error
   #MC_Home_Instance(Axis := "输入轴驱动伺服", Execute := #"Step" = 1, Done => #Temp[0]);   // MC_Home
   IF #Temp[0] THEN #"Step" := 2; END_IF;
END_REGION

REGION Network 4
   #CTRL_HSC_0_Instance(HSC := 1, CV := #"Step" = 1);   // CTRL_HSC
END_REGION

REGION Network 5
   // ENO of a box is taken as its EN; it also drops when the box reports an error
   #MC_Home_Instance_1(Axis := "输入轴移载伺服", Execute := #"Step" = 2, Mode := 3, Done => #Temp[1]);   // MC_Home
   IF #Temp[1] THEN #"Step" := 3; END_IF;
END_REGION

REGION Network 6
   #_w1 := #"Step" = 3;
   IF #_w1 THEN
       "输出轴花键移载气缸退" := TRUE;
       "输出轴花键移载气缸进" := FALSE;
   END_IF;
   #IEC_Timer_0_Instance(IN := #_w1 AND "输出轴花键移载气缸退", PT := T#1s);   // TON
   IF #IEC_Timer_0_Instance.Q THEN
       #"Step" := 4;
       "输出轴花键移载气缸退" := FALSE;
   END_IF;
END_REGION

REGION Network 7
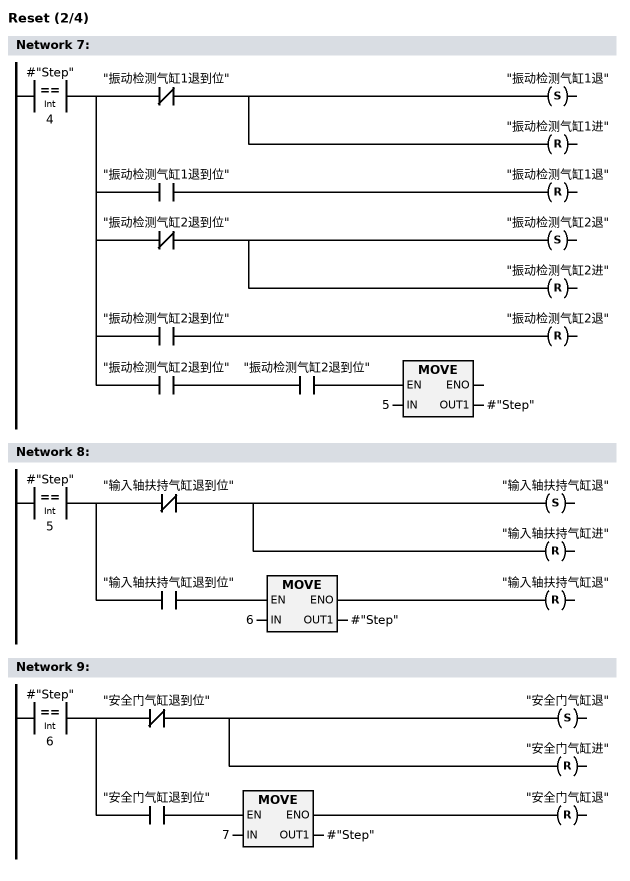
   RUNG wire#powerrail
      { S7_Templates := "SrcType := Int" } EQ_Contact(in1 := #"Step", in2 := 4)
      wire#w1
      I_Contact( "振动检测气缸1退到位" )
      wire#w2
      S_Coil( "振动检测气缸1退" )
   END_RUNG
   RUNG wire#w2
      R_Coil( "振动检测气缸1进" )
   END_RUNG
   RUNG wire#w1
      Contact( "振动检测气缸1退到位" )
      R_Coil( "振动检测气缸1退" )
   END_RUNG
   RUNG wire#w1
      I_Contact( "振动检测气缸2退到位" )
      wire#w3
      S_Coil( "振动检测气缸2退" )
   END_RUNG
   RUNG wire#w3
      R_Coil( "振动检测气缸2进" )
   END_RUNG
   RUNG wire#w1
      Contact( "振动检测气缸2退到位" )
      R_Coil( "振动检测气缸2退" )
   END_RUNG
   RUNG wire#w1
      Contact( "振动检测气缸2退到位" )
      Contact( "振动检测气缸2退到位" )
      Move(in := 5, out1 => #"Step")
   END_RUNG
   // the same network as SCL:
   #_w1 := #"Step" = 4;
   IF #_w1 AND NOT "振动检测气缸1退到位" THEN
       "振动检测气缸1退" := TRUE;
       "振动检测气缸1进" := FALSE;
   END_IF;
   IF #_w1 AND "振动检测气缸1退到位" THEN "振动检测气缸1退" := FALSE; END_IF;
   IF #_w1 AND NOT "振动检测气缸2退到位" THEN
       "振动检测气缸2退" := TRUE;
       "振动检测气缸2进" := FALSE;
   END_IF;
   IF #_w1 AND "振动检测气缸2退到位" THEN "振动检测气缸2退" := FALSE; END_IF;
   IF #_w1 AND "振动检测气缸2退到位" AND "振动检测气缸2退到位" THEN #"Step" := 5; END_IF;
END_REGION

REGION Network 8
   RUNG wire#powerrail
      { S7_Templates := "SrcType := Int" } EQ_Contact(in1 := #"Step", in2 := 5)
      wire#w1
      I_Contact( "输入轴扶持气缸退到位" )
      wire#w2
      S_Coil( "输入轴扶持气缸退" )
   END_RUNG
   RUNG wire#w2
      R_Coil( "输入轴扶持气缸进" )
   END_RUNG
   RUNG wire#w1
      Contact( "输入轴扶持气缸退到位" )
      Move(in := 6, out1 => #"Step")
      R_Coil( "输入轴扶持气缸退" )
   END_RUNG
   // the same network as SCL:
   #_w1 := #"Step" = 5;
   IF #_w1 AND NOT "输入轴扶持气缸退到位" THEN
       "输入轴扶持气缸退" := TRUE;
       "输入轴扶持气缸进" := FALSE;
   END_IF;
   IF #_w1 AND "输入轴扶持气缸退到位" THEN
       #"Step" := 6;
       "输入轴扶持气缸退" := FALSE;
   END_IF;
END_REGION

REGION Network 9
   RUNG wire#powerrail
      { S7_Templates := "SrcType := Int" } EQ_Contact(in1 := #"Step", in2 := 6)
      wire#w1
      I_Contact( "安全门气缸退到位" )
      wire#w2
      S_Coil( "安全门气缸退" )
   END_RUNG
   RUNG wire#w2
      R_Coil( "安全门气缸进" )
   END_RUNG
   RUNG wire#w1
      Contact( "安全门气缸退到位" )
      Move(in := 7, out1 => #"Step")
      R_Coil( "安全门气缸退" )
   END_RUNG
   // the same network as SCL:
   #_w1 := #"Step" = 6;
   IF #_w1 AND NOT "安全门气缸退到位" THEN
       "安全门气缸退" := TRUE;
       "安全门气缸进" := FALSE;
   END_IF;
   IF #_w1 AND "安全门气缸退到位" THEN
       #"Step" := 7;
       "安全门气缸退" := FALSE;
   END_IF;
END_REGION

REGION Network 10
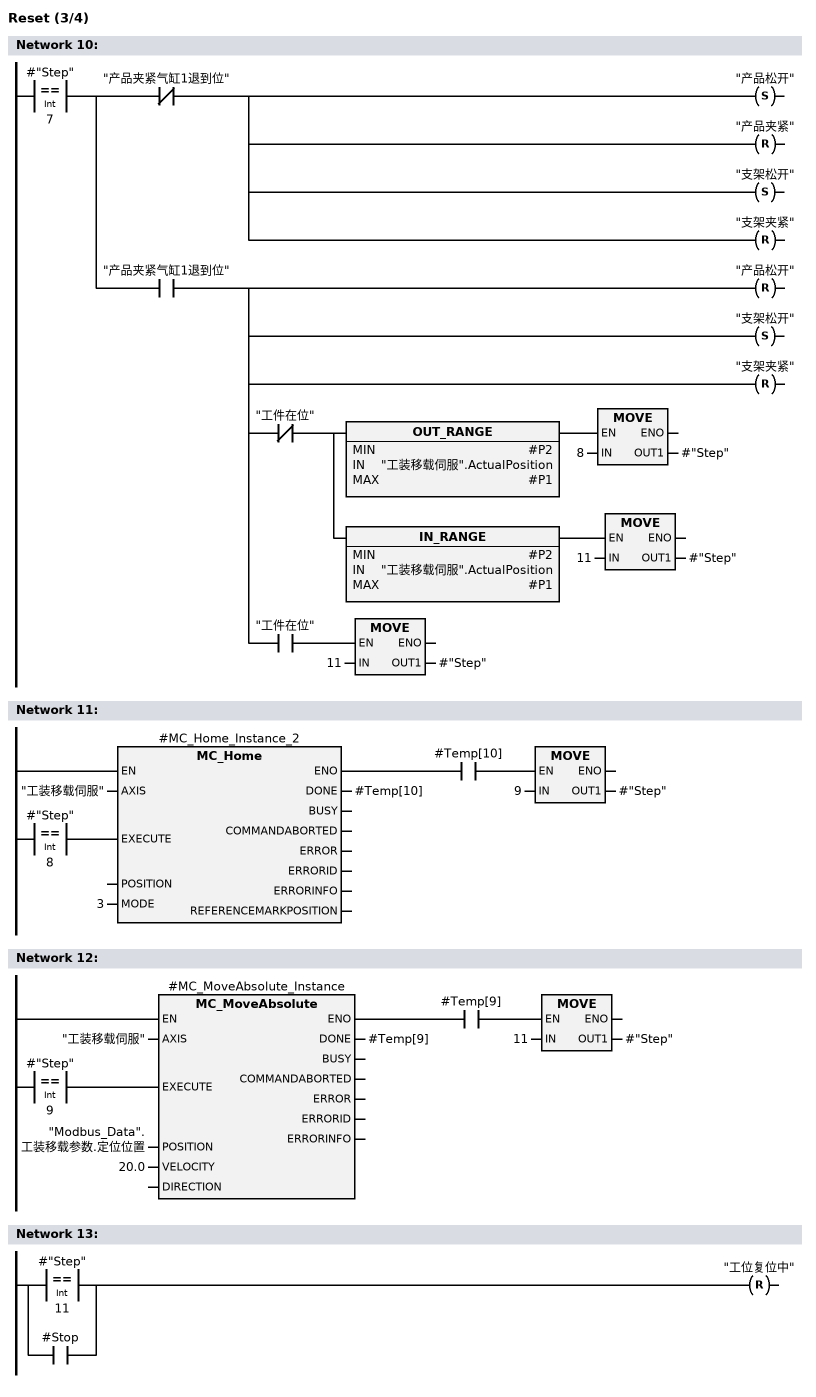
   #_w1 := #"Step" = 7;
   IF #_w1 AND NOT "产品夹紧气缸1退到位" THEN
       "产品松开" := TRUE;
       "产品夹紧" := FALSE;
       "支架松开" := TRUE;
       "支架夹紧" := FALSE;
   END_IF;
   #_w2 := #_w1 AND "产品夹紧气缸1退到位";
   IF #_w2 THEN
       "产品松开" := FALSE;
       "支架松开" := TRUE;
       "支架夹紧" := FALSE;
   END_IF;
   #_w3 := #_w2 AND NOT "工件在位";
   IF #_w3 AND (("工装移载伺服".ActualPosition < #P2) OR ("工装移载伺服".ActualPosition > #P1)) THEN
       #"Step" := 8;
   END_IF;
   IF #_w3 AND (#P2 <= "工装移载伺服".ActualPosition) AND ("工装移载伺服".ActualPosition <= #P1) THEN
       #"Step" := 11;
   END_IF;
   IF #_w2 AND "工件在位" THEN #"Step" := 11; END_IF;
END_REGION

REGION Network 11
   // ENO of a box is taken as its EN; it also drops when the box reports an error
   #MC_Home_Instance_2(Axis := "工装移载伺服", Execute := #"Step" = 8, Mode := 3, Done => #Temp[10]);   // MC_Home
   IF #Temp[10] THEN #"Step" := 9; END_IF;
END_REGION

REGION Network 12
   // ENO of a box is taken as its EN; it also drops when the box reports an error
   #MC_MoveAbsolute_Instance(Axis := "工装移载伺服",   // MC_MoveAbsolute
                           Execute := #"Step" = 9,
                           Position := "Modbus_Data".工装移载参数.定位位置,
                           Velocity := 20.0,
                           Done => #Temp[9]);
   IF #Temp[9] THEN #"Step" := 11; END_IF;
END_REGION

REGION Network 13
   RUNG wire#powerrail
      { S7_Templates := "SrcType := Int" } EQ_Contact(in1 := #"Step", in2 := 11)
      wire#w1
      R_Coil( "工位复位中" )
   END_RUNG
   RUNG wire#powerrail
      Contact( #Stop )
   END_RUNG wire#w1
   // the same network as SCL:
   IF (#"Step" = 11) OR #Stop THEN "工位复位中" := FALSE; END_IF;
END_REGION

REGION Network 14
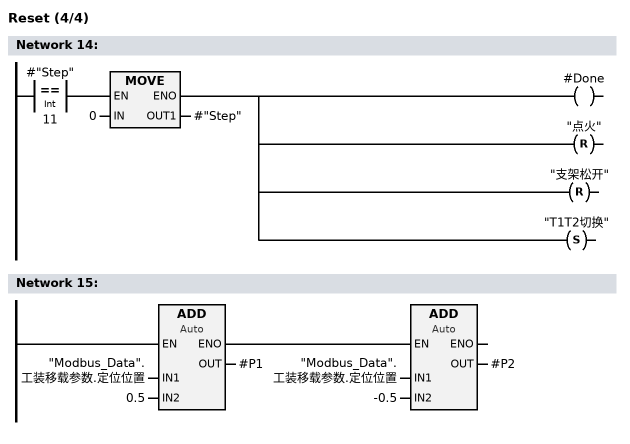
   RUNG wire#powerrail
      { S7_Templates := "SrcType := Int" } EQ_Contact(in1 := #"Step", in2 := 11)
      Move(in := 0, out1 => #"Step")
      wire#w1
      Coil( #Done )
   END_RUNG
   RUNG wire#w1
      R_Coil( "点火" )
   END_RUNG
   RUNG wire#w1
      R_Coil( "支架松开" )
   END_RUNG
   RUNG wire#w1
      S_Coil( "T1T2切换" )
   END_RUNG
   // the same network as SCL:
   #_w1 := #"Step" = 11;
   IF #_w1 THEN #"Step" := 0; END_IF;
   #Done := #_w1;
   IF #_w1 THEN
       "点火" := FALSE;
       "支架松开" := FALSE;
       "T1T2切换" := TRUE;
   END_IF;
END_REGION

REGION Network 15
   RUNG wire#powerrail
      Add(in1 := "Modbus_Data".工装移载参数.定位位置, in2 := 0.5, out => #P1)
      Add(in1 := "Modbus_Data".工装移载参数.定位位置, in2 := -0.5, out => #P2)
   END_RUNG
   // the same network as SCL:
   #P1 := "Modbus_Data".工装移载参数.定位位置 + 0.5;
   #P2 := "Modbus_Data".工装移载参数.定位位置 + (-0.5);
END_REGION
END_FUNCTION_BLOCK

FUNCTION_BLOCK "Alarm"   // FB5, LAD
{ S7_Optimized_Access := 'TRUE' }
VERSION : 0.1
   VAR
      "Step" : Int;
      Temp : Array[0..7] of Bool;
      IEC_Timer_0_Instance : TON_TIME;
      IEC_Timer_0_Instance_1 : TON_TIME;
      IEC_Timer_0_Instance_2 : TON_TIME;
      Error_id : Word;
      "Time" : Time := T#5000ms;
      IEC_Timer_0_Instance_3 : TON_TIME;
      IEC_Timer_0_Instance_4 : TON_TIME;
      IEC_Timer_0_Instance_5 : TON_TIME;
      IEC_Timer_0_Instance_6 : TON_TIME;
      IEC_Timer_0_Instance_7 : TON_TIME;
      IEC_Timer_0_Instance_8 : TON_TIME;
      IEC_Timer_0_Instance_9 : TON_TIME;
      IEC_Timer_0_Instance_10 : TON_TIME;
      IEC_Timer_0_Instance_11 : TON_TIME;
      IEC_Timer_0_Instance_12 : TON_TIME;
      IEC_Timer_0_Instance_13 : TON_TIME;
      IEC_Timer_0_Instance_14 : TON_TIME;
      IEC_Timer_0_Instance_15 : TON_TIME;
      IEC_Timer_0_Instance_16 : TON_TIME;
      IEC_Timer_0_Instance_17 : TP_TIME;
      IEC_Timer_0_Instance_18 : TP_TIME;
      IEC_Timer_0_Instance_19 : TON_TIME;
   END_VAR
   VAR_TEMP   // added for the SCL form of the ladder/FBD networks
      _w1 : Bool;
      _w2 : Bool;
   END_VAR
BEGIN

REGION Network 1
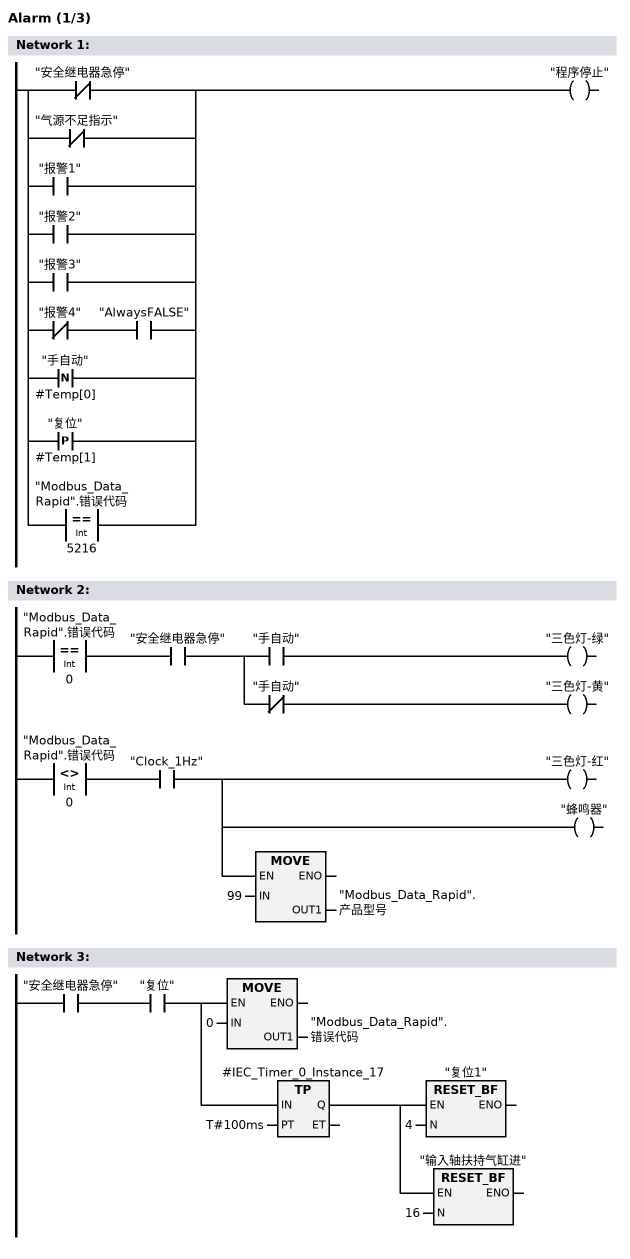
   RUNG wire#powerrail
      I_Contact( "安全继电器急停" )
      wire#w1
      Coil( "程序停止" )
   END_RUNG
   RUNG wire#powerrail
      I_Contact( "气源不足指示" )
   END_RUNG wire#w1
   RUNG wire#powerrail
      Contact( "报警1" )
   END_RUNG wire#w1
   RUNG wire#powerrail
      Contact( "报警2" )
   END_RUNG wire#w1
   RUNG wire#powerrail
      Contact( "报警3" )
   END_RUNG wire#w1
   RUNG wire#powerrail
      I_Contact( "报警4" )
      Contact( "AlwaysFALSE" )
   END_RUNG wire#w1
   RUNG wire#powerrail
      N_Contact(operand := "手自动", bit := #Temp[0])
   END_RUNG wire#w1
   RUNG wire#powerrail
      P_Contact(operand := "复位", bit := #Temp[1])
   END_RUNG wire#w1
   RUNG wire#powerrail
      { S7_Templates := "SrcType := Int" } EQ_Contact(in1 := "Modbus_Data_Rapid".错误代码, in2 := 5216)
   END_RUNG wire#w1
   // the same network as SCL:
   #_w1 := NOT "手自动" AND #Temp[0];   // falling edge of "手自动"
   #Temp[0] := "手自动";
   #_w2 := "复位" AND NOT #Temp[1];   // rising edge of "复位"
   #Temp[1] := "复位";
   "程序停止" := NOT "安全继电器急停" OR NOT "气源不足指示" OR "报警1" OR "报警2" OR "报警3" OR (NOT "报警4" AND "AlwaysFALSE") OR #_w1 OR #_w2 OR ("Modbus_Data_Rapid".错误代码 = 5216);
END_REGION

REGION Network 2
   RUNG wire#powerrail
      { S7_Templates := "SrcType := Int" } EQ_Contact(in1 := "Modbus_Data_Rapid".错误代码, in2 := 0)
      Contact( "安全继电器急停" )
      wire#w1
      Contact( "手自动" )
      Coil( "三色灯-绿" )
   END_RUNG
   RUNG wire#w1
      I_Contact( "手自动" )
      Coil( "三色灯-黄" )
   END_RUNG
   RUNG wire#powerrail
      { S7_Templates := "SrcType := Int" } NE_Contact(in1 := "Modbus_Data_Rapid".错误代码, in2 := 0)
      Contact( "Clock_1Hz" )
      wire#w2
      Coil( "三色灯-红" )
   END_RUNG
   RUNG wire#w2
      Coil( "蜂鸣器" )
   END_RUNG
   RUNG wire#w2
      Move(in := 99, out1 => "Modbus_Data_Rapid".产品型号)
   END_RUNG
   // the same network as SCL:
   #_w1 := ("Modbus_Data_Rapid".错误代码 = 0) AND "安全继电器急停";
   "三色灯-绿" := #_w1 AND "手自动";
   "三色灯-黄" := #_w1 AND NOT "手自动";
   "三色灯-红" := ("Modbus_Data_Rapid".错误代码 <> 0) AND "Clock_1Hz";
   "蜂鸣器" := "三色灯-红";
   IF "三色灯-红" THEN "Modbus_Data_Rapid".产品型号 := 99; END_IF;
END_REGION

REGION Network 3
   // no SCL statement known for RBitfield: written as a call
   #_w1 := "安全继电器急停" AND "复位";
   IF #_w1 THEN "Modbus_Data_Rapid".错误代码 := 0; END_IF;
   #IEC_Timer_0_Instance_17(IN := #_w1, PT := T#100ms);   // TP
   IF #IEC_Timer_0_Instance_17.Q THEN
       RESET_BF(operand := "复位1", n := 4);
       RESET_BF(operand := "输入轴扶持气缸进", n := 16);
   END_IF;
END_REGION

REGION Network 4
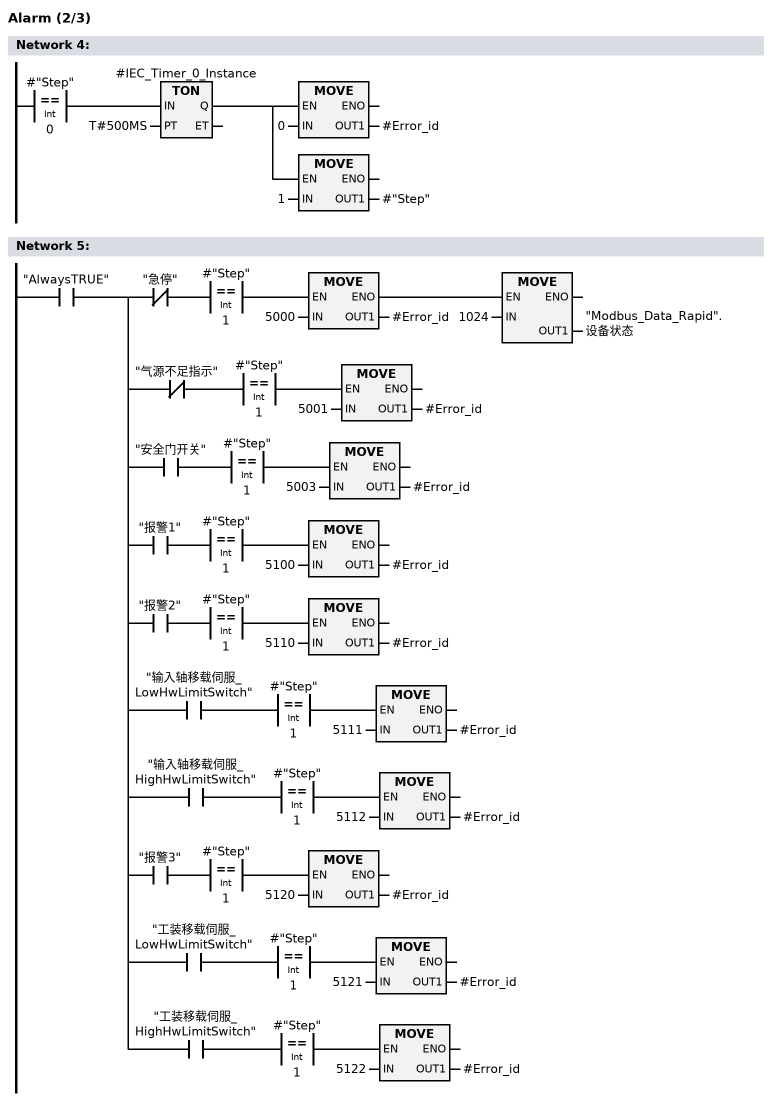
   #IEC_Timer_0_Instance(IN := #"Step" = 0, PT := T#500MS);   // TON
   IF #IEC_Timer_0_Instance.Q THEN
       #Error_id := 0;
       #"Step" := 1;
   END_IF;
END_REGION

REGION Network 5
   RUNG wire#powerrail
      Contact( "AlwaysTRUE" )
      wire#w1
      I_Contact( "急停" )
      { S7_Templates := "SrcType := Int" } EQ_Contact(in1 := #"Step", in2 := 1)
      Move(in := 5000, out1 => #Error_id)
      Move(in := 1024, out1 => "Modbus_Data_Rapid".设备状态)
   END_RUNG
   RUNG wire#w1
      I_Contact( "气源不足指示" )
      { S7_Templates := "SrcType := Int" } EQ_Contact(in1 := #"Step", in2 := 1)
      Move(in := 5001, out1 => #Error_id)
   END_RUNG
   RUNG wire#w1
      Contact( "安全门开关" )
      { S7_Templates := "SrcType := Int" } EQ_Contact(in1 := #"Step", in2 := 1)
      Move(in := 5003, out1 => #Error_id)
   END_RUNG
   RUNG wire#w1
      Contact( "报警1" )
      { S7_Templates := "SrcType := Int" } EQ_Contact(in1 := #"Step", in2 := 1)
      Move(in := 5100, out1 => #Error_id)
   END_RUNG
   RUNG wire#w1
      Contact( "报警2" )
      { S7_Templates := "SrcType := Int" } EQ_Contact(in1 := #"Step", in2 := 1)
      Move(in := 5110, out1 => #Error_id)
   END_RUNG
   RUNG wire#w1
      Contact( "输入轴移载伺服_LowHwLimitSwitch" )
      { S7_Templates := "SrcType := Int" } EQ_Contact(in1 := #"Step", in2 := 1)
      Move(in := 5111, out1 => #Error_id)
   END_RUNG
   RUNG wire#w1
      Contact( "输入轴移载伺服_HighHwLimitSwitch" )
      { S7_Templates := "SrcType := Int" } EQ_Contact(in1 := #"Step", in2 := 1)
      Move(in := 5112, out1 => #Error_id)
   END_RUNG
   RUNG wire#w1
      Contact( "报警3" )
      { S7_Templates := "SrcType := Int" } EQ_Contact(in1 := #"Step", in2 := 1)
      Move(in := 5120, out1 => #Error_id)
   END_RUNG
   RUNG wire#w1
      Contact( "工装移载伺服_LowHwLimitSwitch" )
      { S7_Templates := "SrcType := Int" } EQ_Contact(in1 := #"Step", in2 := 1)
      Move(in := 5121, out1 => #Error_id)
   END_RUNG
   RUNG wire#w1
      Contact( "工装移载伺服_HighHwLimitSwitch" )
      { S7_Templates := "SrcType := Int" } EQ_Contact(in1 := #"Step", in2 := 1)
      Move(in := 5122, out1 => #Error_id)
   END_RUNG
   // the same network as SCL:
   IF "AlwaysTRUE" AND NOT "急停" AND (#"Step" = 1) THEN
       #Error_id := 5000;
       "Modbus_Data_Rapid".设备状态 := 1024;
   END_IF;
   IF "AlwaysTRUE" AND NOT "气源不足指示" AND (#"Step" = 1) THEN #Error_id := 5001; END_IF;
   IF "AlwaysTRUE" AND "安全门开关" AND (#"Step" = 1) THEN #Error_id := 5003; END_IF;
   IF "AlwaysTRUE" AND "报警1" AND (#"Step" = 1) THEN #Error_id := 5100; END_IF;
   IF "AlwaysTRUE" AND "报警2" AND (#"Step" = 1) THEN #Error_id := 5110; END_IF;
   IF "AlwaysTRUE" AND "输入轴移载伺服_LowHwLimitSwitch" AND (#"Step" = 1) THEN #Error_id := 5111; END_IF;
   IF "AlwaysTRUE" AND "输入轴移载伺服_HighHwLimitSwitch" AND (#"Step" = 1) THEN #Error_id := 5112; END_IF;
   IF "AlwaysTRUE" AND "报警3" AND (#"Step" = 1) THEN #Error_id := 5120; END_IF;
   IF "AlwaysTRUE" AND "工装移载伺服_LowHwLimitSwitch" AND (#"Step" = 1) THEN #Error_id := 5121; END_IF;
   IF "AlwaysTRUE" AND "工装移载伺服_HighHwLimitSwitch" AND (#"Step" = 1) THEN #Error_id := 5122; END_IF;
END_REGION

REGION Network 6
   // 到位故障
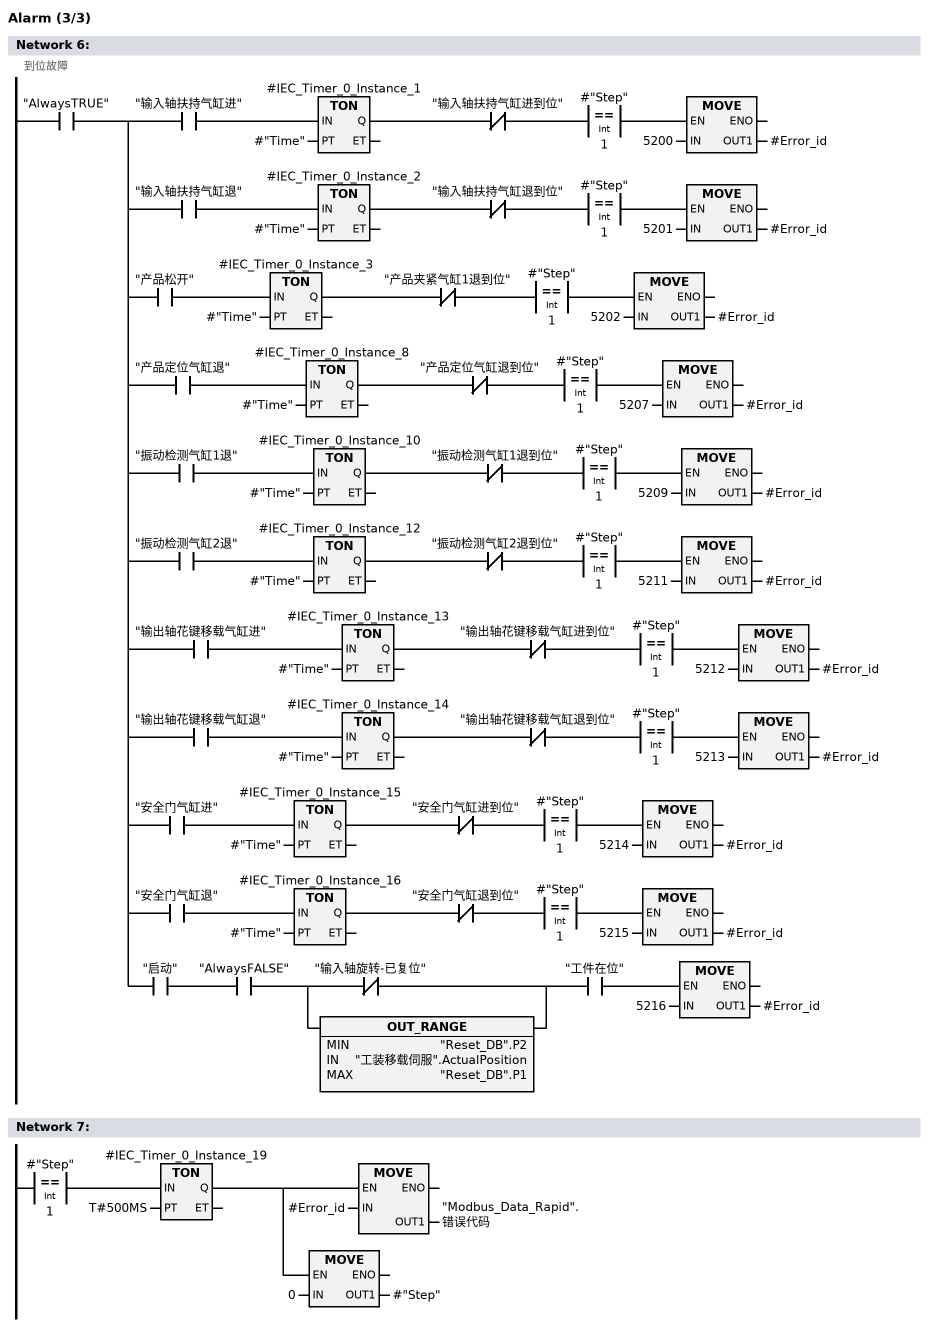
   #IEC_Timer_0_Instance_1(IN := "AlwaysTRUE" AND "输入轴扶持气缸进", PT := #"Time");   // TON
   IF #IEC_Timer_0_Instance_1.Q AND NOT "输入轴扶持气缸进到位" AND (#"Step" = 1) THEN #Error_id := 5200; END_IF;
   #IEC_Timer_0_Instance_2(IN := "AlwaysTRUE" AND "输入轴扶持气缸退", PT := #"Time");   // TON
   IF #IEC_Timer_0_Instance_2.Q AND NOT "输入轴扶持气缸退到位" AND (#"Step" = 1) THEN #Error_id := 5201; END_IF;
   #IEC_Timer_0_Instance_3(IN := "AlwaysTRUE" AND "产品松开", PT := #"Time");   // TON
   IF #IEC_Timer_0_Instance_3.Q AND NOT "产品夹紧气缸1退到位" AND (#"Step" = 1) THEN #Error_id := 5202; END_IF;
   #IEC_Timer_0_Instance_8(IN := "AlwaysTRUE" AND "产品定位气缸退", PT := #"Time");   // TON
   IF #IEC_Timer_0_Instance_8.Q AND NOT "产品定位气缸退到位" AND (#"Step" = 1) THEN #Error_id := 5207; END_IF;
   #IEC_Timer_0_Instance_10(IN := "AlwaysTRUE" AND "振动检测气缸1退", PT := #"Time");   // TON
   IF #IEC_Timer_0_Instance_10.Q AND NOT "振动检测气缸1退到位" AND (#"Step" = 1) THEN #Error_id := 5209; END_IF;
   #IEC_Timer_0_Instance_12(IN := "AlwaysTRUE" AND "振动检测气缸2退", PT := #"Time");   // TON
   IF #IEC_Timer_0_Instance_12.Q AND NOT "振动检测气缸2退到位" AND (#"Step" = 1) THEN #Error_id := 5211; END_IF;
   #IEC_Timer_0_Instance_13(IN := "AlwaysTRUE" AND "输出轴花键移载气缸进", PT := #"Time");   // TON
   IF #IEC_Timer_0_Instance_13.Q AND NOT "输出轴花键移载气缸进到位" AND (#"Step" = 1) THEN #Error_id := 5212; END_IF;
   #IEC_Timer_0_Instance_14(IN := "AlwaysTRUE" AND "输出轴花键移载气缸退", PT := #"Time");   // TON
   IF #IEC_Timer_0_Instance_14.Q AND NOT "输出轴花键移载气缸退到位" AND (#"Step" = 1) THEN #Error_id := 5213; END_IF;
   #IEC_Timer_0_Instance_15(IN := "AlwaysTRUE" AND "安全门气缸进", PT := #"Time");   // TON
   IF #IEC_Timer_0_Instance_15.Q AND NOT "安全门气缸进到位" AND (#"Step" = 1) THEN #Error_id := 5214; END_IF;
   #IEC_Timer_0_Instance_16(IN := "AlwaysTRUE" AND "安全门气缸退", PT := #"Time");   // TON
   IF #IEC_Timer_0_Instance_16.Q AND NOT "安全门气缸退到位" AND (#"Step" = 1) THEN #Error_id := 5215; END_IF;
   IF "AlwaysTRUE" AND "启动" AND "AlwaysFALSE" AND (NOT "输入轴旋转-已复位" OR ("工装移载伺服".ActualPosition < "Reset_DB".P2) OR ("工装移载伺服".ActualPosition > "Reset_DB".P1)) AND "工件在位" THEN
       #Error_id := 5216;
   END_IF;
END_REGION

REGION Network 7
   #IEC_Timer_0_Instance_19(IN := #"Step" = 1, PT := T#500MS);   // TON
   IF #IEC_Timer_0_Instance_19.Q THEN
       "Modbus_Data_Rapid".错误代码 := #Error_id;
       #"Step" := 0;
   END_IF;
END_REGION
END_FUNCTION_BLOCK

FUNCTION_BLOCK "套花键"   // FB6, LAD
{ S7_Optimized_Access := 'TRUE' }
VERSION : 0.1
   VAR_INPUT
      Axis_In : TO_PositioningAxis;
      Axis_In_Sway : TO_PositioningAxis;
      Parameter : "In_config";
      Axis_Position : Real;
      Excute : Bool;
      Stop : Bool;
   END_VAR
   VAR_OUTPUT
      Done : Bool;
      Error : Bool;
      Busy : Bool;
   END_VAR
   VAR
      "Step" : Int;
      Temp : Array[0..7] of Bool;
      MC_MoveAbsolute_Instance : MC_MoveAbsolute;
      MC_MoveAbsolute_Instance_1 : MC_MoveAbsolute;
      左右摆动_Instance : "左右摆动";
   END_VAR
   VAR_TEMP
      done1 : Bool;
      done2 : Bool;
      done3 : Bool;
      done4 : Bool;
      n : Bool;
      n_1 : Bool;
      lang : Real;
   END_VAR
   VAR_TEMP   // added for the SCL form of the ladder/FBD networks
      _w1 : Bool;
      _w2 : Bool;
   END_VAR
BEGIN

REGION Network 1
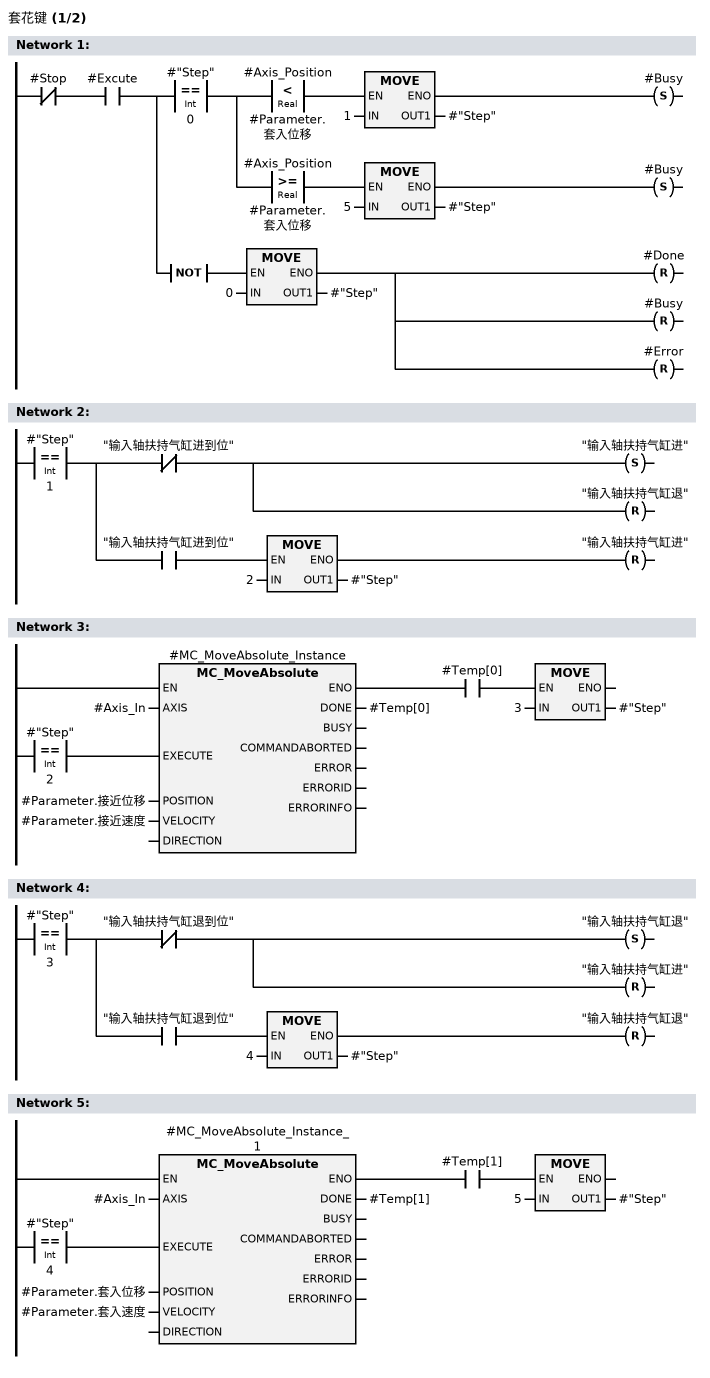
   RUNG wire#powerrail
      I_Contact( #Stop )
      Contact( #Excute )
      wire#w1
      { S7_Templates := "SrcType := Int" } EQ_Contact(in1 := #"Step", in2 := 0)
      wire#w2
      { S7_Templates := "SrcType := Real" } LT_Contact(in1 := #Axis_Position, in2 := #Parameter.套入位移)
      Move(in := 1, out1 => #"Step")
      S_Coil( #Busy )
   END_RUNG
   RUNG wire#w2
      { S7_Templates := "SrcType := Real" } GE_Contact(in1 := #Axis_Position, in2 := #Parameter.套入位移)
      Move(in := 5, out1 => #"Step")
      S_Coil( #Busy )
   END_RUNG
   RUNG wire#w1
      Not()
      Move(in := 0, out1 => #"Step")
      wire#w3
      R_Coil( #Done )
   END_RUNG
   RUNG wire#w3
      R_Coil( #Busy )
   END_RUNG
   RUNG wire#w3
      R_Coil( #Error )
   END_RUNG
   // the same network as SCL:
   #_w1 := NOT #Stop AND #Excute;
   #_w2 := #_w1 AND (#"Step" = 0);
   IF #_w2 AND (#Axis_Position < #Parameter.套入位移) THEN
       #"Step" := 1;
       #Busy := TRUE;
   END_IF;
   IF #_w2 AND (#Axis_Position >= #Parameter.套入位移) THEN
       #"Step" := 5;
       #Busy := TRUE;
   END_IF;
   IF NOT #_w1 THEN
       #"Step" := 0;
       #Done := FALSE;
       #Busy := FALSE;
       #Error := FALSE;
   END_IF;
END_REGION

REGION Network 2
   RUNG wire#powerrail
      { S7_Templates := "SrcType := Int" } EQ_Contact(in1 := #"Step", in2 := 1)
      wire#w1
      I_Contact( "输入轴扶持气缸进到位" )
      wire#w2
      S_Coil( "输入轴扶持气缸进" )
   END_RUNG
   RUNG wire#w2
      R_Coil( "输入轴扶持气缸退" )
   END_RUNG
   RUNG wire#w1
      Contact( "输入轴扶持气缸进到位" )
      Move(in := 2, out1 => #"Step")
      R_Coil( "输入轴扶持气缸进" )
   END_RUNG
   // the same network as SCL:
   #_w1 := #"Step" = 1;
   IF #_w1 AND NOT "输入轴扶持气缸进到位" THEN
       "输入轴扶持气缸进" := TRUE;
       "输入轴扶持气缸退" := FALSE;
   END_IF;
   IF #_w1 AND "输入轴扶持气缸进到位" THEN
       #"Step" := 2;
       "输入轴扶持气缸进" := FALSE;
   END_IF;
END_REGION

REGION Network 3
   // ENO of a box is taken as its EN; it also drops when the box reports an error
   #MC_MoveAbsolute_Instance(Axis := #Axis_In,   // MC_MoveAbsolute
                           Execute := #"Step" = 2,
                           Position := #Parameter.接近位移,
                           Velocity := #Parameter.接近速度,
                           Done => #Temp[0]);
   IF #Temp[0] THEN #"Step" := 3; END_IF;
END_REGION

REGION Network 4
   RUNG wire#powerrail
      { S7_Templates := "SrcType := Int" } EQ_Contact(in1 := #"Step", in2 := 3)
      wire#w1
      I_Contact( "输入轴扶持气缸退到位" )
      wire#w2
      S_Coil( "输入轴扶持气缸退" )
   END_RUNG
   RUNG wire#w2
      R_Coil( "输入轴扶持气缸进" )
   END_RUNG
   RUNG wire#w1
      Contact( "输入轴扶持气缸退到位" )
      Move(in := 4, out1 => #"Step")
      R_Coil( "输入轴扶持气缸退" )
   END_RUNG
   // the same network as SCL:
   #_w1 := #"Step" = 3;
   IF #_w1 AND NOT "输入轴扶持气缸退到位" THEN
       "输入轴扶持气缸退" := TRUE;
       "输入轴扶持气缸进" := FALSE;
   END_IF;
   IF #_w1 AND "输入轴扶持气缸退到位" THEN
       #"Step" := 4;
       "输入轴扶持气缸退" := FALSE;
   END_IF;
END_REGION

REGION Network 5
   // ENO of a box is taken as its EN; it also drops when the box reports an error
   #MC_MoveAbsolute_Instance_1(Axis := #Axis_In,   // MC_MoveAbsolute
                           Execute := #"Step" = 4,
                           Position := #Parameter.套入位移,
                           Velocity := #Parameter.套入速度,
                           Done => #Temp[1]);
   IF #Temp[1] THEN #"Step" := 5; END_IF;
END_REGION

REGION Network 6
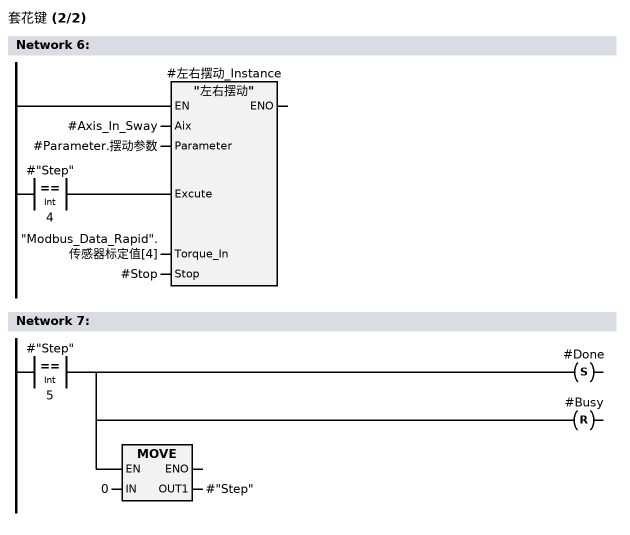
   RUNG wire#powerrail
      #左右摆动_Instance(Excute := wire#w1, Aix := #Axis_In_Sway, Parameter := #Parameter.摆动参数, Torque_In := "Modbus_Data_Rapid".传感器标定值[4], Stop := #Stop)
   END_RUNG
   RUNG wire#powerrail
      { S7_Templates := "SrcType := Int" } EQ_Contact(in1 := #"Step", in2 := 4)
   END_RUNG wire#w1
   // the same network as SCL:
   #左右摆动_Instance(Aix := #Axis_In_Sway,   // "左右摆动"
                  Parameter := #Parameter.摆动参数,
                  Excute := #"Step" = 4,
                  Torque_In := "Modbus_Data_Rapid".传感器标定值[4],
                  Stop := #Stop);
END_REGION

REGION Network 7
   RUNG wire#powerrail
      { S7_Templates := "SrcType := Int" } EQ_Contact(in1 := #"Step", in2 := 5)
      wire#w1
      S_Coil( #Done )
   END_RUNG
   RUNG wire#w1
      R_Coil( #Busy )
   END_RUNG
   RUNG wire#w1
      Move(in := 0, out1 => #"Step")
   END_RUNG
   // the same network as SCL:
   IF #"Step" = 5 THEN
       #Done := TRUE;
       #Busy := FALSE;
       #"Step" := 0;
   END_IF;
END_REGION
END_FUNCTION_BLOCK

FUNCTION_BLOCK "功能"   // FB7, LAD
{ S7_Optimized_Access := 'TRUE' }
VERSION : 0.1
   VAR_INPUT
      Aix_In : TO_PositioningAxis;
      Parameter : "Test_Function_CFG";
      Excute : Bool;
      Dir : Bool;
      Torque_In : Real;
      Stop : Bool;
   END_VAR
   VAR_OUTPUT
      Done : Bool;
      Busy : Bool;
      Error : Bool;
   END_VAR
   VAR
      "Step" : Int;
      Protection_Torque : Real;
      Function_Angle : Real;
      Temp : Array[0..7] of Bool;
      MC_Halt_Instance : MC_Halt;
      MC_Halt_Instance_1 : MC_Halt;
      MC_Home_Instance_1 : MC_Home;
      MC_MoveRelative_Instance_1 : MC_MoveRelative;
      MC_MoveRelative_Instance_2 : MC_MoveRelative;
      MC_Halt_Instance_2 : MC_Halt;
      MC_MoveAbsolute_Instance : MC_MoveAbsolute;
      IEC_Timer_0_Instance : TON_TIME;
   END_VAR
   VAR_TEMP   // added for the SCL form of the ladder/FBD networks
      _w1 : Bool;
   END_VAR
BEGIN

REGION Network 1
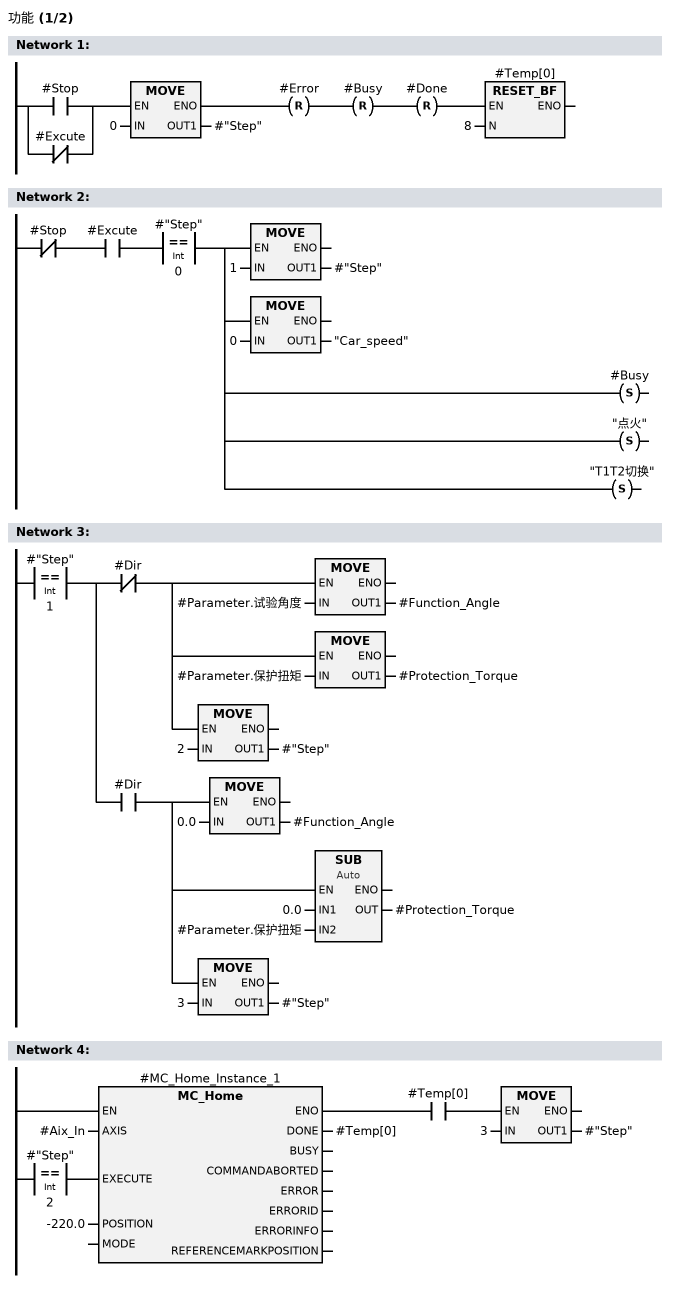
   // no SCL statement known for RBitfield: written as a call
   IF #Stop OR NOT #Excute THEN
       #"Step" := 0;
       #Error := FALSE;
       #Busy := FALSE;
       #Done := FALSE;
       RESET_BF(operand := #Temp[0], n := 8);
   END_IF;
END_REGION

REGION Network 2
   RUNG wire#powerrail
      I_Contact( #Stop )
      Contact( #Excute )
      { S7_Templates := "SrcType := Int" } EQ_Contact(in1 := #"Step", in2 := 0)
      wire#w1
      Move(in := 1, out1 => #"Step")
   END_RUNG
   RUNG wire#w1
      Move(in := 0, out1 => "Car_speed")
   END_RUNG
   RUNG wire#w1
      S_Coil( #Busy )
   END_RUNG
   RUNG wire#w1
      S_Coil( "点火" )
   END_RUNG
   RUNG wire#w1
      S_Coil( "T1T2切换" )
   END_RUNG
   // the same network as SCL:
   #_w1 := NOT #Stop AND #Excute AND (#"Step" = 0);
   IF #_w1 THEN
       #"Step" := 1;
       "Car_speed" := 0;
       #Busy := TRUE;
       "点火" := TRUE;
       "T1T2切换" := TRUE;
   END_IF;
END_REGION

REGION Network 3
   RUNG wire#powerrail
      { S7_Templates := "SrcType := Int" } EQ_Contact(in1 := #"Step", in2 := 1)
      wire#w1
      I_Contact( #Dir )
      wire#w2
      Move(in := #Parameter.试验角度, out1 => #Function_Angle)
   END_RUNG
   RUNG wire#w2
      Move(in := #Parameter.保护扭矩, out1 => #Protection_Torque)
   END_RUNG
   RUNG wire#w2
      Move(in := 2, out1 => #"Step")
   END_RUNG
   RUNG wire#w1
      Contact( #Dir )
      wire#w3
      Move(in := 0.0, out1 => #Function_Angle)
   END_RUNG
   RUNG wire#w3
      Sub(in1 := 0.0, in2 := #Parameter.保护扭矩, out => #Protection_Torque)
   END_RUNG
   RUNG wire#w3
      Move(in := 3, out1 => #"Step")
   END_RUNG
   // the same network as SCL:
   #_w1 := #"Step" = 1;
   IF #_w1 AND NOT #Dir THEN
       #Function_Angle := #Parameter.试验角度;
       #Protection_Torque := #Parameter.保护扭矩;
       #"Step" := 2;
   END_IF;
   IF #_w1 AND #Dir THEN
       #Function_Angle := 0.0;
       #Protection_Torque := 0.0 - #Parameter.保护扭矩;
       #"Step" := 3;
   END_IF;
END_REGION

REGION Network 4
   // ENO of a box is taken as its EN; it also drops when the box reports an error
   #MC_Home_Instance_1(Axis := #Aix_In, Execute := #"Step" = 2, Position := -220.0, Done => #Temp[0]);   // MC_Home
   IF #Temp[0] THEN #"Step" := 3; END_IF;
END_REGION

REGION Network 5
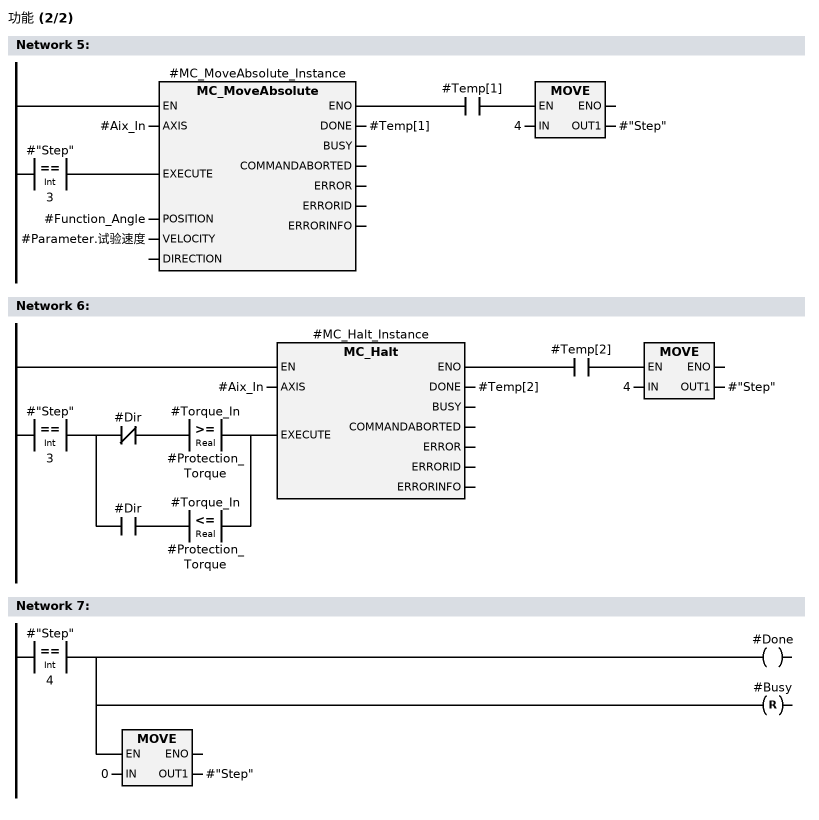
   // ENO of a box is taken as its EN; it also drops when the box reports an error
   #MC_MoveAbsolute_Instance(Axis := #Aix_In,   // MC_MoveAbsolute
                           Execute := #"Step" = 3,
                           Position := #Function_Angle,
                           Velocity := #Parameter.试验速度,
                           Done => #Temp[1]);
   IF #Temp[1] THEN #"Step" := 4; END_IF;
END_REGION

REGION Network 6
   // ENO of a box is taken as its EN; it also drops when the box reports an error
   #MC_Halt_Instance(Axis := #Aix_In,   // MC_Halt
                     Execute := (#"Step" = 3) AND ((NOT #Dir AND (#Torque_In >= #Protection_Torque)) OR (#Dir AND (#Torque_In <= #Protection_Torque))),
                     Done => #Temp[2]);
   IF #Temp[2] THEN #"Step" := 4; END_IF;
END_REGION

REGION Network 7
   RUNG wire#powerrail
      { S7_Templates := "SrcType := Int" } EQ_Contact(in1 := #"Step", in2 := 4)
      wire#w1
      Coil( #Done )
   END_RUNG
   RUNG wire#w1
      R_Coil( #Busy )
   END_RUNG
   RUNG wire#w1
      Move(in := 0, out1 => #"Step")
   END_RUNG
   // the same network as SCL:
   #Done := #"Step" = 4;
   IF #Done THEN
       #Busy := FALSE;
       #"Step" := 0;
   END_IF;
END_REGION
END_FUNCTION_BLOCK

FUNCTION_BLOCK "左右摆动"   // FB8, LAD
{ S7_Optimized_Access := 'TRUE' }
VERSION : 0.1
   VAR_INPUT
      Aix : TO_PositioningAxis;
      Parameter : "In_swing_config";
      Excute : Bool;
      Torque_In : Real;
      Stop : Bool;
   END_VAR
   VAR
      "Step" : Int;
      Protection_Torque_N : Real;
      Swing_Angle_N : Real;
      Temp : Array[0..7] of Bool;
      MC_Halt_Instance : MC_Halt;
      MC_Home_Instance : MC_Home;
      MC_Halt_Instance_1 : MC_Halt;
      MC_Halt_Instance_2 : MC_Halt;
      MC_MoveAbsolute_Instance : MC_MoveAbsolute;
      MC_MoveAbsolute_Instance_1 : MC_MoveAbsolute;
      MC_MoveJog_Instance : MC_MoveJog;
      IEC_Timer_0_Instance : TON_TIME;
      IEC_Timer_0_Instance_1 : TON_TIME;
      MC_MoveRelative_Instance : MC_MoveRelative;
      MC_MoveRelative_Instance_1 : MC_MoveRelative;
      MC_Halt_Instance_3 : MC_Halt;
      MC_Halt_Instance_4 : MC_Halt;
      MC_Home_Instance_1 : MC_Home;
   END_VAR
   VAR_TEMP   // added for the SCL form of the ladder/FBD networks
      _w1 : Bool;
   END_VAR
BEGIN

REGION Network 1
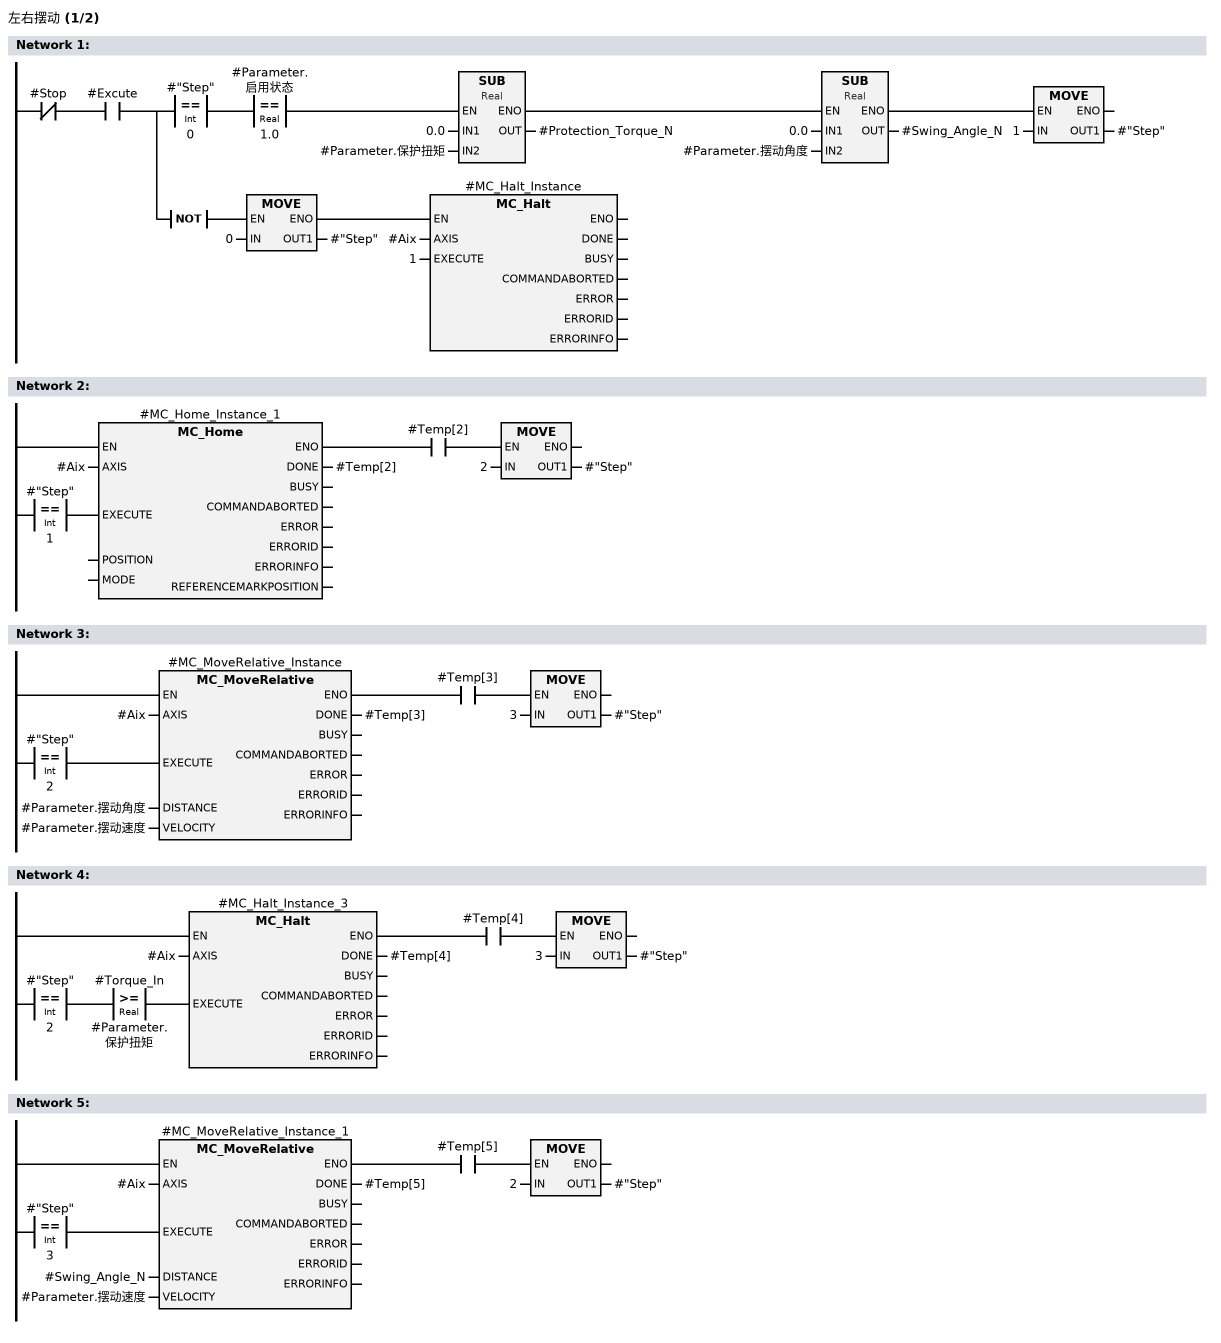
   #_w1 := NOT #Stop AND #Excute;
   IF #_w1 AND (#"Step" = 0) AND (#Parameter.启用状态 = 1.0) THEN
       #Protection_Torque_N := 0.0 - #Parameter.保护扭矩;
       #Swing_Angle_N := 0.0 - #Parameter.摆动角度;
       #"Step" := 1;
   END_IF;
   IF NOT #_w1 THEN
       #"Step" := 0;
       #MC_Halt_Instance(Axis := #Aix, Execute := 1);   // MC_Halt
   END_IF;
END_REGION

REGION Network 2
   // ENO of a box is taken as its EN; it also drops when the box reports an error
   #MC_Home_Instance_1(Axis := #Aix, Execute := #"Step" = 1, Done => #Temp[2]);   // MC_Home
   IF #Temp[2] THEN #"Step" := 2; END_IF;
END_REGION

REGION Network 3
   // ENO of a box is taken as its EN; it also drops when the box reports an error
   #MC_MoveRelative_Instance(Axis := #Aix,   // MC_MoveRelative
                           Execute := #"Step" = 2,
                           Distance := #Parameter.摆动角度,
                           Velocity := #Parameter.摆动速度,
                           Done => #Temp[3]);
   IF #Temp[3] THEN #"Step" := 3; END_IF;
END_REGION

REGION Network 4
   // ENO of a box is taken as its EN; it also drops when the box reports an error
   #MC_Halt_Instance_3(Axis := #Aix,   // MC_Halt
                       Execute := (#"Step" = 2) AND (#Torque_In >= #Parameter.保护扭矩),
                       Done => #Temp[4]);
   IF #Temp[4] THEN #"Step" := 3; END_IF;
END_REGION

REGION Network 5
   // ENO of a box is taken as its EN; it also drops when the box reports an error
   #MC_MoveRelative_Instance_1(Axis := #Aix,   // MC_MoveRelative
                           Execute := #"Step" = 3,
                           Distance := #Swing_Angle_N,
                           Velocity := #Parameter.摆动速度,
                           Done => #Temp[5]);
   IF #Temp[5] THEN #"Step" := 2; END_IF;
END_REGION

REGION Network 6
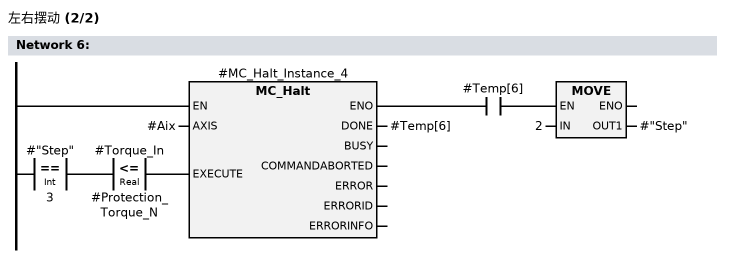
   // ENO of a box is taken as its EN; it also drops when the box reports an error
   #MC_Halt_Instance_4(Axis := #Aix,   // MC_Halt
                       Execute := (#"Step" = 3) AND (#Torque_In <= #Protection_Torque_N),
                       Done => #Temp[6]);
   IF #Temp[6] THEN #"Step" := 2; END_IF;
END_REGION
END_FUNCTION_BLOCK

FUNCTION_BLOCK "空载"   // FB9, LAD
{ S7_Optimized_Access := 'TRUE' }
VERSION : 0.1
   VAR_INPUT
      Aix_In : TO_PositioningAxis;
      Parameter : "Test_No_Load_CFG";
      Excute : Bool;
      Dir : Bool;
      Torque_In : Real;
      Stop : Bool;
   END_VAR
   VAR_OUTPUT
      Done : Bool;
      Busy : Bool;
      Error : Bool;
   END_VAR
   VAR
      "Step" : Int;
      Protection_Torque : Real;
      NoLoad_Angle : Real;
      Temp : Array[0..7] of Bool;
      MC_Halt_Instance : MC_Halt;
      MC_Home_Instance : MC_Home;
      MC_MoveAbsolute_Instance : MC_MoveAbsolute;
   END_VAR
   VAR_TEMP   // added for the SCL form of the ladder/FBD networks
      _w1 : Bool;
      _w2 : Bool;
   END_VAR
BEGIN

REGION Network 1
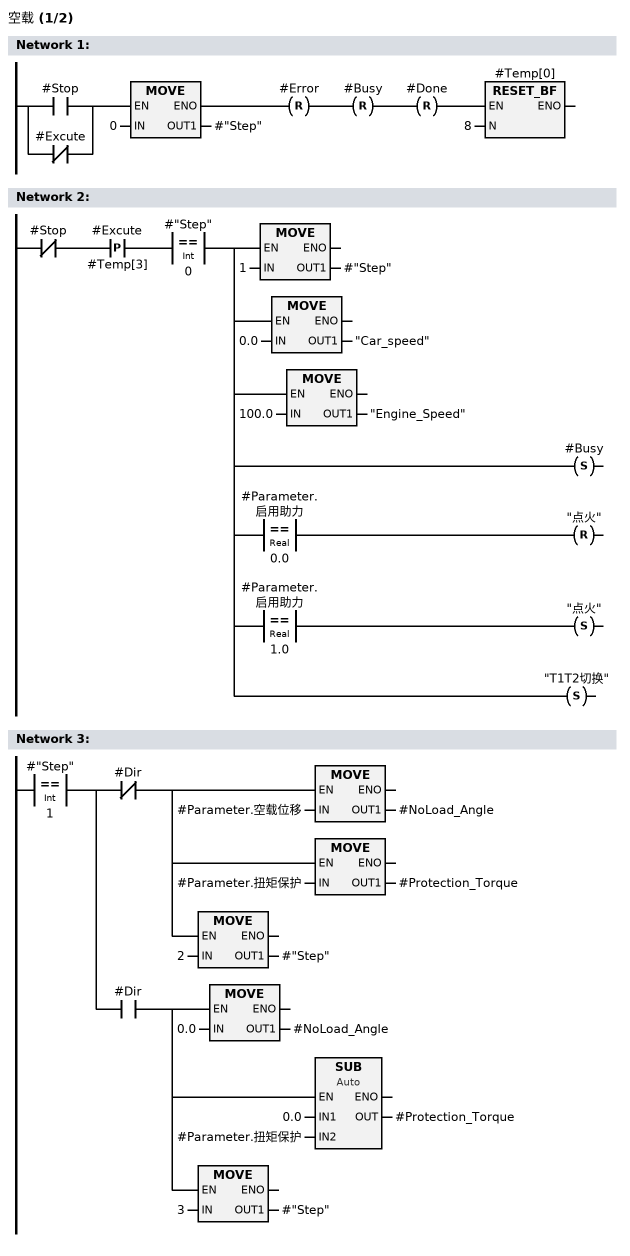
   // no SCL statement known for RBitfield: written as a call
   IF #Stop OR NOT #Excute THEN
       #"Step" := 0;
       #Error := FALSE;
       #Busy := FALSE;
       #Done := FALSE;
       RESET_BF(operand := #Temp[0], n := 8);
   END_IF;
END_REGION

REGION Network 2
   RUNG wire#powerrail
      I_Contact( #Stop )
      P_Contact(operand := #Excute, bit := #Temp[3])
      { S7_Templates := "SrcType := Int" } EQ_Contact(in1 := #"Step", in2 := 0)
      wire#w1
      Move(in := 1, out1 => #"Step")
   END_RUNG
   RUNG wire#w1
      Move(in := 0.0, out1 => "Car_speed")
   END_RUNG
   RUNG wire#w1
      Move(in := 100.0, out1 => "Engine_Speed")
   END_RUNG
   RUNG wire#w1
      S_Coil( #Busy )
   END_RUNG
   RUNG wire#w1
      { S7_Templates := "SrcType := Real" } EQ_Contact(in1 := #Parameter.启用助力, in2 := 0.0)
      R_Coil( "点火" )
   END_RUNG
   RUNG wire#w1
      { S7_Templates := "SrcType := Real" } EQ_Contact(in1 := #Parameter.启用助力, in2 := 1.0)
      S_Coil( "点火" )
   END_RUNG
   RUNG wire#w1
      S_Coil( "T1T2切换" )
   END_RUNG
   // the same network as SCL:
   #_w1 := NOT #Stop AND #Excute AND NOT #Temp[3];   // rising edge of #Excute
   #Temp[3] := #Excute;
   #_w2 := #_w1 AND (#"Step" = 0);
   IF #_w2 THEN
       #"Step" := 1;
       "Car_speed" := 0.0;
       "Engine_Speed" := 100.0;
       #Busy := TRUE;
   END_IF;
   IF #_w2 AND (#Parameter.启用助力 = 0.0) THEN "点火" := FALSE; END_IF;
   IF #_w2 AND (#Parameter.启用助力 = 1.0) THEN "点火" := TRUE; END_IF;
   IF #_w2 THEN "T1T2切换" := TRUE; END_IF;
END_REGION

REGION Network 3
   RUNG wire#powerrail
      { S7_Templates := "SrcType := Int" } EQ_Contact(in1 := #"Step", in2 := 1)
      wire#w1
      I_Contact( #Dir )
      wire#w2
      Move(in := #Parameter.空载位移, out1 => #NoLoad_Angle)
   END_RUNG
   RUNG wire#w2
      Move(in := #Parameter.扭矩保护, out1 => #Protection_Torque)
   END_RUNG
   RUNG wire#w2
      Move(in := 2, out1 => #"Step")
   END_RUNG
   RUNG wire#w1
      Contact( #Dir )
      wire#w3
      Move(in := 0.0, out1 => #NoLoad_Angle)
   END_RUNG
   RUNG wire#w3
      Sub(in1 := 0.0, in2 := #Parameter.扭矩保护, out => #Protection_Torque)
   END_RUNG
   RUNG wire#w3
      Move(in := 3, out1 => #"Step")
   END_RUNG
   // the same network as SCL:
   #_w1 := #"Step" = 1;
   IF #_w1 AND NOT #Dir THEN
       #NoLoad_Angle := #Parameter.空载位移;
       #Protection_Torque := #Parameter.扭矩保护;
       #"Step" := 2;
   END_IF;
   IF #_w1 AND #Dir THEN
       #NoLoad_Angle := 0.0;
       #Protection_Torque := 0.0 - #Parameter.扭矩保护;
       #"Step" := 3;
   END_IF;
END_REGION

REGION Network 4
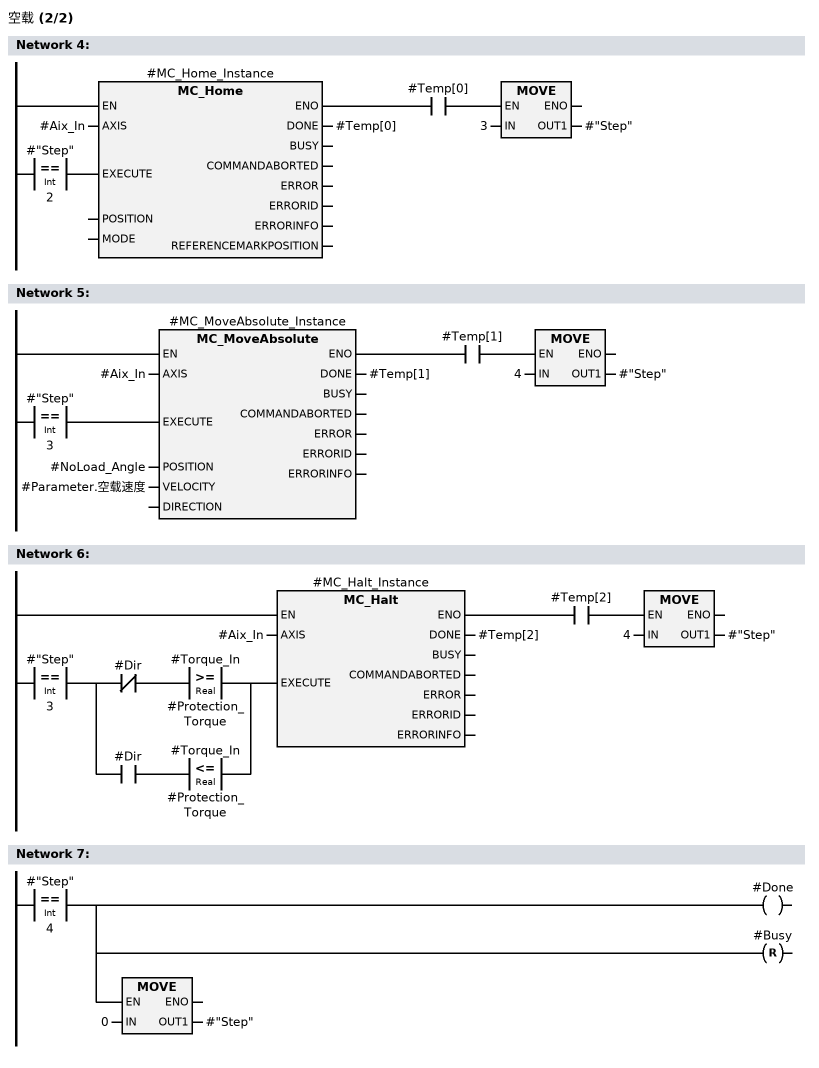
   // ENO of a box is taken as its EN; it also drops when the box reports an error
   #MC_Home_Instance(Axis := #Aix_In, Execute := #"Step" = 2, Done => #Temp[0]);   // MC_Home
   IF #Temp[0] THEN #"Step" := 3; END_IF;
END_REGION

REGION Network 5
   // ENO of a box is taken as its EN; it also drops when the box reports an error
   #MC_MoveAbsolute_Instance(Axis := #Aix_In,   // MC_MoveAbsolute
                           Execute := #"Step" = 3,
                           Position := #NoLoad_Angle,
                           Velocity := #Parameter.空载速度,
                           Done => #Temp[1]);
   IF #Temp[1] THEN #"Step" := 4; END_IF;
END_REGION

REGION Network 6
   // ENO of a box is taken as its EN; it also drops when the box reports an error
   #MC_Halt_Instance(Axis := #Aix_In,   // MC_Halt
                     Execute := (#"Step" = 3) AND ((NOT #Dir AND (#Torque_In >= #Protection_Torque)) OR (#Dir AND (#Torque_In <= #Protection_Torque))),
                     Done => #Temp[2]);
   IF #Temp[2] THEN #"Step" := 4; END_IF;
END_REGION

REGION Network 7
   RUNG wire#powerrail
      { S7_Templates := "SrcType := Int" } EQ_Contact(in1 := #"Step", in2 := 4)
      wire#w1
      Coil( #Done )
   END_RUNG
   RUNG wire#w1
      R_Coil( #Busy )
   END_RUNG
   RUNG wire#w1
      Move(in := 0, out1 => #"Step")
   END_RUNG
   // the same network as SCL:
   #Done := #"Step" = 4;
   IF #Done THEN
       #Busy := FALSE;
       #"Step" := 0;
   END_IF;
END_REGION
END_FUNCTION_BLOCK

FUNCTION_BLOCK "Auto"   // FB10, LAD
{ S7_Optimized_Access := 'TRUE' }
VERSION : 0.1
   VAR
      Temp : Array[0..15] of Bool;
      套花键_Instance : "套花键";
      空载_Instance : "空载";
      空载_Instance_1 : "空载";
      功能_Instance : "功能";
      功能_Instance_1 : "功能";
      力特性_Instance : "力特性";
      力特性_Instance_1 : "力特性";
      力特性_Instance_2 : "力特性";
      力特性_Instance_3 : "力特性";
      振动_Instance : "振动";
      振动_Instance_1 : "振动";
      MC_MoveAbsolute_Instance : MC_MoveAbsolute;
      IEC_Timer_0_Instance : TOF_TIME;
      IEC_Timer_0_Instance_1 : TOF_TIME;
      IEC_Timer_0_Instance_2 : TOF_TIME;
      IEC_Timer_0_Instance_3 : TOF_TIME;
      IEC_Timer_0_Instance_4 : TOF_TIME;
      IEC_Timer_0_Instance_5 : TOF_TIME;
      IEC_Timer_0_Instance_6 : TOF_TIME;
      IEC_Timer_0_Instance_7 : TOF_TIME;
      IEC_Timer_0_Instance_8 : TOF_TIME;
      IEC_Timer_0_Instance_9 : TOF_TIME;
      力特性_Instance_4 : "力特性";
      力特性_Instance_5 : "力特性";
      IEC_Timer_0_Instance_10 : TON_TIME;
      IEC_Timer_0_Instance_11 : TOF_TIME;
      IEC_Timer_0_Instance_12 : TON_TIME;
   END_VAR
   VAR_TEMP   // added for the SCL form of the ladder/FBD networks
      _w1 : Bool;
   END_VAR
BEGIN

REGION Network 1
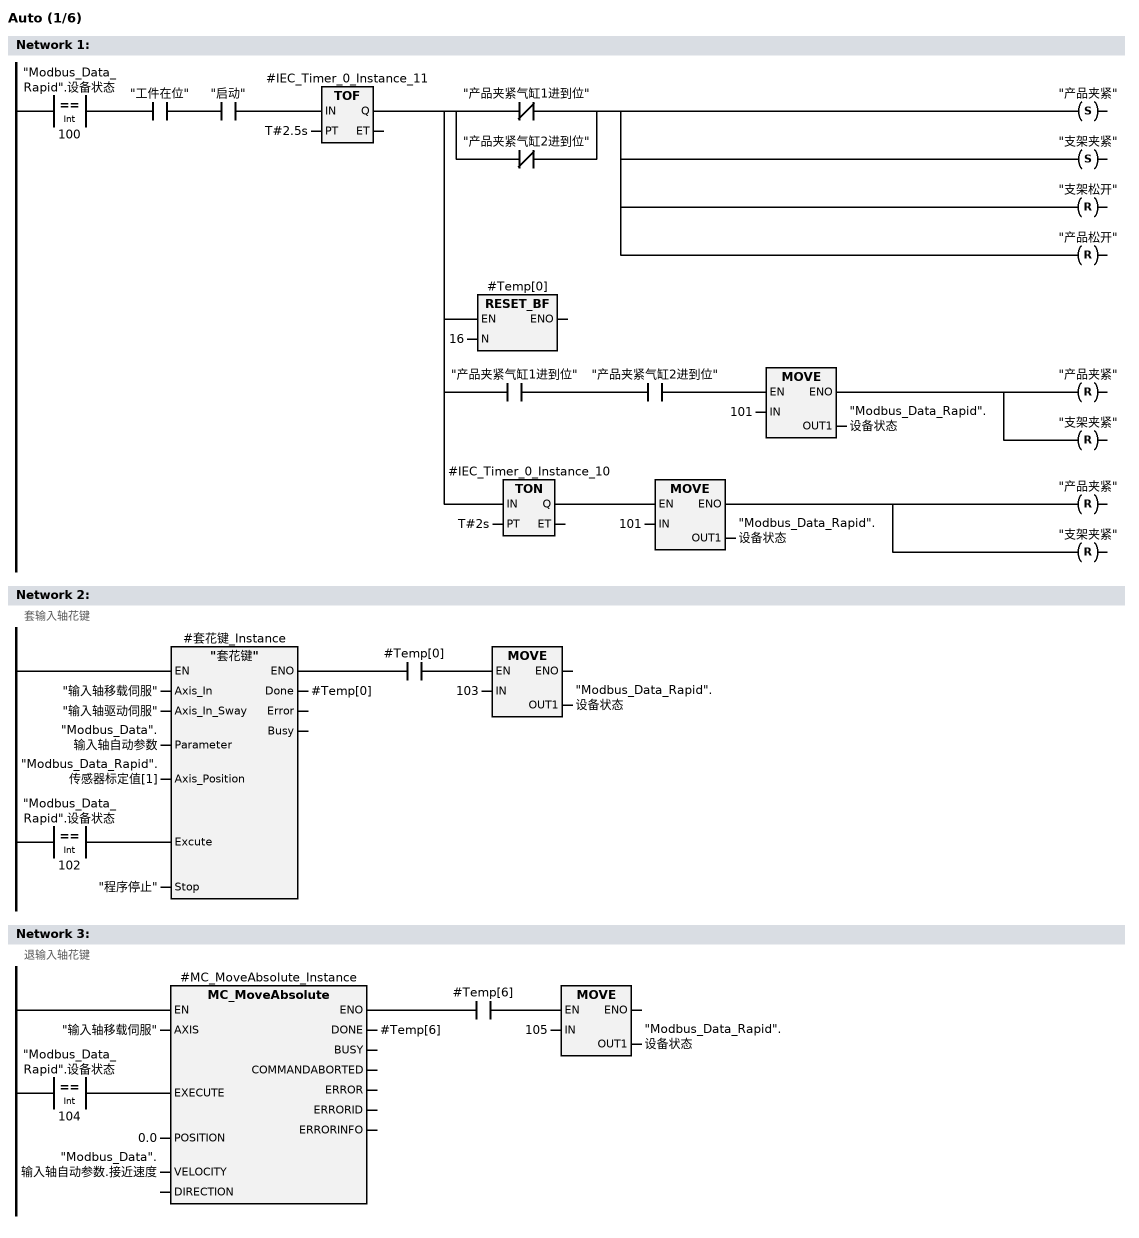
   // no SCL statement known for RBitfield: written as a call
   #IEC_Timer_0_Instance_11(IN := ("Modbus_Data_Rapid".设备状态 = 100) AND "工件在位" AND "启动", PT := T#2.5s);   // TOF
   IF #IEC_Timer_0_Instance_11.Q AND (NOT "产品夹紧气缸1进到位" OR NOT "产品夹紧气缸2进到位") THEN
       "产品夹紧" := TRUE;
       "支架夹紧" := TRUE;
       "支架松开" := FALSE;
       "产品松开" := FALSE;
   END_IF;
   IF #IEC_Timer_0_Instance_11.Q THEN RESET_BF(operand := #Temp[0], n := 16); END_IF;
   IF #IEC_Timer_0_Instance_11.Q AND "产品夹紧气缸1进到位" AND "产品夹紧气缸2进到位" THEN
       "Modbus_Data_Rapid".设备状态 := 101;
       "产品夹紧" := FALSE;
       "支架夹紧" := FALSE;
   END_IF;
   #IEC_Timer_0_Instance_10(IN := #IEC_Timer_0_Instance_11.Q, PT := T#2s);   // TON
   IF #IEC_Timer_0_Instance_10.Q THEN
       "Modbus_Data_Rapid".设备状态 := 101;
       "产品夹紧" := FALSE;
       "支架夹紧" := FALSE;
   END_IF;
END_REGION

REGION Network 2
   // 套输入轴花键
   RUNG wire#powerrail
      #套花键_Instance(Excute := wire#w1, Axis_In := "输入轴移载伺服", Axis_In_Sway := "输入轴驱动伺服", Parameter := "Modbus_Data".输入轴自动参数, Axis_Position := "Modbus_Data_Rapid".传感器标定值[1], Stop := "程序停止", Done => #Temp[0], Error =>, Busy =>)
      Contact( #Temp[0] )
      Move(in := 103, out1 => "Modbus_Data_Rapid".设备状态)
   END_RUNG
   RUNG wire#powerrail
      { S7_Templates := "SrcType := Int" } EQ_Contact(in1 := "Modbus_Data_Rapid".设备状态, in2 := 102)
   END_RUNG wire#w1
   // the same network as SCL:
   #套花键_Instance(Axis_In := "输入轴移载伺服",   // "套花键"
                 Axis_In_Sway := "输入轴驱动伺服",
                 Parameter := "Modbus_Data".输入轴自动参数,
                 Axis_Position := "Modbus_Data_Rapid".传感器标定值[1],
                 Excute := "Modbus_Data_Rapid".设备状态 = 102,
                 Stop := "程序停止",
                 Done => #Temp[0],
                 ENO => #_w1);
   IF #_w1 AND #Temp[0] THEN "Modbus_Data_Rapid".设备状态 := 103; END_IF;
END_REGION

REGION Network 3
   // 退输入轴花键
   // ENO of a box is taken as its EN; it also drops when the box reports an error
   #MC_MoveAbsolute_Instance(Axis := "输入轴移载伺服",   // MC_MoveAbsolute
                           Execute := "Modbus_Data_Rapid".设备状态 = 104,
                           Position := 0.0,
                           Velocity := "Modbus_Data".输入轴自动参数.接近速度,
                           Done => #Temp[6]);
   IF #Temp[6] THEN "Modbus_Data_Rapid".设备状态 := 105; END_IF;
END_REGION

REGION Network 4
   // 套输出轴花键
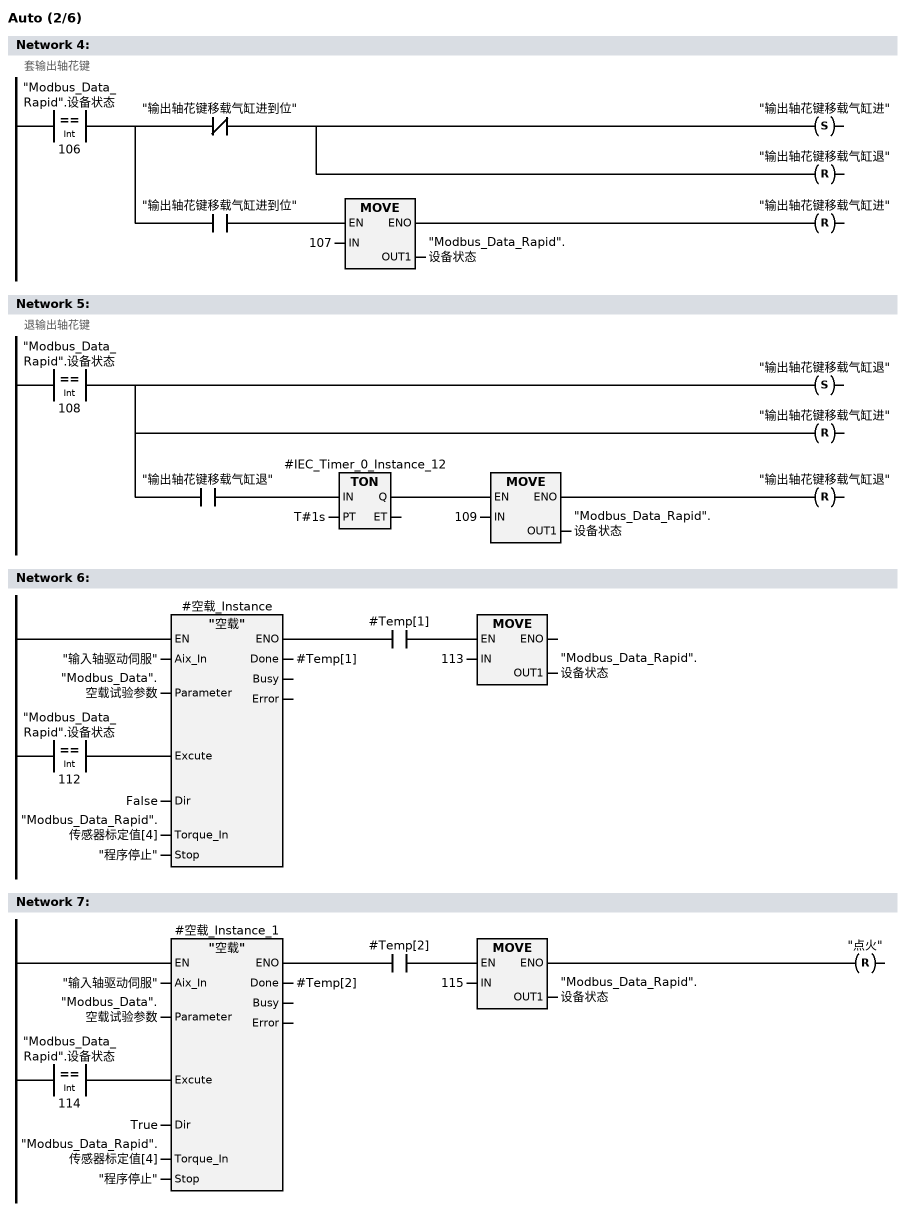
   RUNG wire#powerrail
      { S7_Templates := "SrcType := Int" } EQ_Contact(in1 := "Modbus_Data_Rapid".设备状态, in2 := 106)
      wire#w1
      I_Contact( "输出轴花键移载气缸进到位" )
      wire#w2
      S_Coil( "输出轴花键移载气缸进" )
   END_RUNG
   RUNG wire#w2
      R_Coil( "输出轴花键移载气缸退" )
   END_RUNG
   RUNG wire#w1
      Contact( "输出轴花键移载气缸进到位" )
      Move(in := 107, out1 => "Modbus_Data_Rapid".设备状态)
      R_Coil( "输出轴花键移载气缸进" )
   END_RUNG
   // the same network as SCL:
   #_w1 := "Modbus_Data_Rapid".设备状态 = 106;
   IF #_w1 AND NOT "输出轴花键移载气缸进到位" THEN
       "输出轴花键移载气缸进" := TRUE;
       "输出轴花键移载气缸退" := FALSE;
   END_IF;
   IF #_w1 AND "输出轴花键移载气缸进到位" THEN
       "Modbus_Data_Rapid".设备状态 := 107;
       "输出轴花键移载气缸进" := FALSE;
   END_IF;
END_REGION

REGION Network 5
   // 退输出轴花键
   #_w1 := "Modbus_Data_Rapid".设备状态 = 108;
   IF #_w1 THEN
       "输出轴花键移载气缸退" := TRUE;
       "输出轴花键移载气缸进" := FALSE;
   END_IF;
   #IEC_Timer_0_Instance_12(IN := #_w1 AND "输出轴花键移载气缸退", PT := T#1s);   // TON
   IF #IEC_Timer_0_Instance_12.Q THEN
       "Modbus_Data_Rapid".设备状态 := 109;
       "输出轴花键移载气缸退" := FALSE;
   END_IF;
END_REGION

REGION Network 6
   RUNG wire#powerrail
      #空载_Instance(Excute := wire#w1, Aix_In := "输入轴驱动伺服", Parameter := "Modbus_Data".空载试验参数, Dir := False, Torque_In := "Modbus_Data_Rapid".传感器标定值[4], Stop := "程序停止", Done => #Temp[1], Busy =>, Error =>)
      Contact( #Temp[1] )
      Move(in := 113, out1 => "Modbus_Data_Rapid".设备状态)
   END_RUNG
   RUNG wire#powerrail
      { S7_Templates := "SrcType := Int" } EQ_Contact(in1 := "Modbus_Data_Rapid".设备状态, in2 := 112)
   END_RUNG wire#w1
   // the same network as SCL:
   #空载_Instance(Aix_In := "输入轴驱动伺服",   // "空载"
                Parameter := "Modbus_Data".空载试验参数,
                Excute := "Modbus_Data_Rapid".设备状态 = 112,
                Dir := False,
                Torque_In := "Modbus_Data_Rapid".传感器标定值[4],
                Stop := "程序停止",
                Done => #Temp[1],
                ENO => #_w1);
   IF #_w1 AND #Temp[1] THEN "Modbus_Data_Rapid".设备状态 := 113; END_IF;
END_REGION

REGION Network 7
   RUNG wire#powerrail
      #空载_Instance_1(Excute := wire#w1, Aix_In := "输入轴驱动伺服", Parameter := "Modbus_Data".空载试验参数, Dir := True, Torque_In := "Modbus_Data_Rapid".传感器标定值[4], Stop := "程序停止", Done => #Temp[2], Busy =>, Error =>)
      Contact( #Temp[2] )
      Move(in := 115, out1 => "Modbus_Data_Rapid".设备状态)
      R_Coil( "点火" )
   END_RUNG
   RUNG wire#powerrail
      { S7_Templates := "SrcType := Int" } EQ_Contact(in1 := "Modbus_Data_Rapid".设备状态, in2 := 114)
   END_RUNG wire#w1
   // the same network as SCL:
   #空载_Instance_1(Aix_In := "输入轴驱动伺服",   // "空载"
                  Parameter := "Modbus_Data".空载试验参数,
                  Excute := "Modbus_Data_Rapid".设备状态 = 114,
                  Dir := True,
                  Torque_In := "Modbus_Data_Rapid".传感器标定值[4],
                  Stop := "程序停止",
                  Done => #Temp[2],
                  ENO => #_w1);
   IF #_w1 AND #Temp[2] THEN
       "Modbus_Data_Rapid".设备状态 := 115;
       "点火" := FALSE;
   END_IF;
END_REGION

REGION Network 8
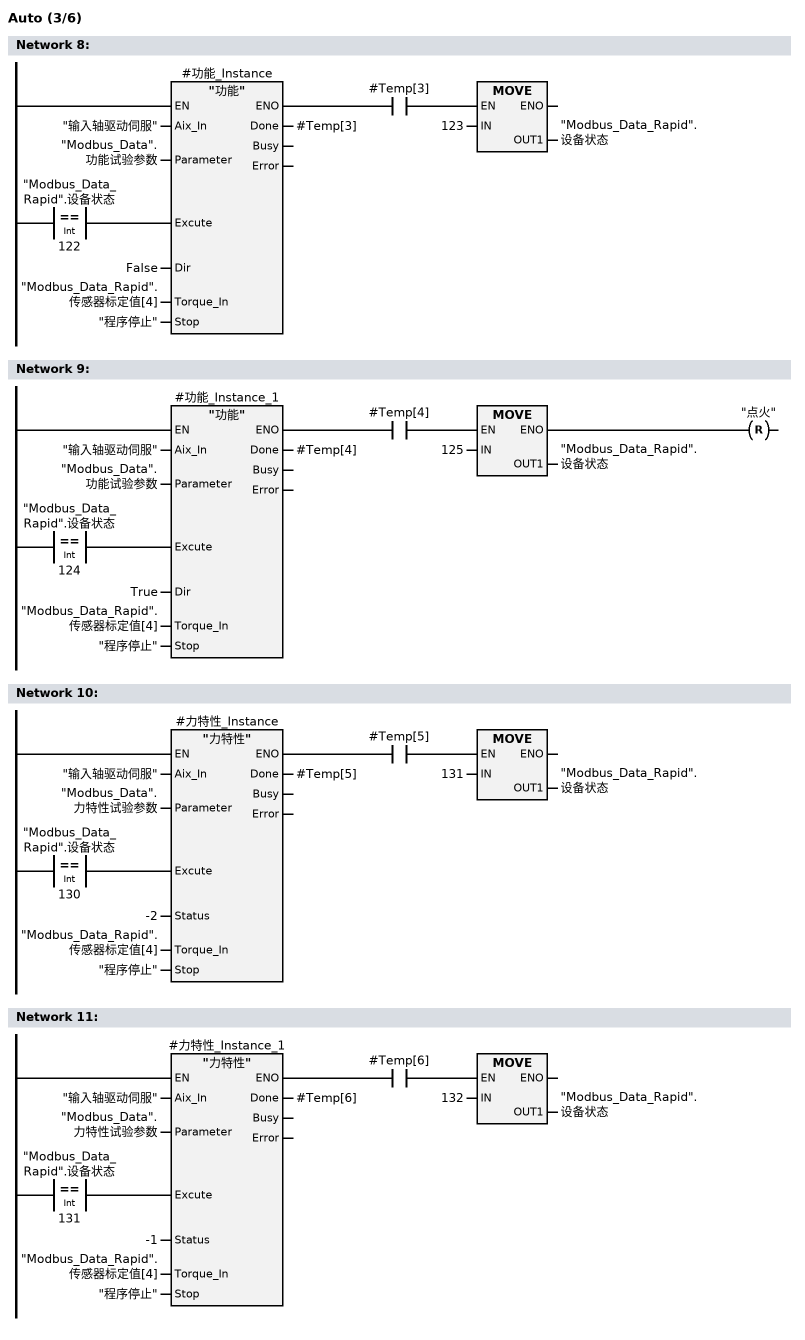
   RUNG wire#powerrail
      #功能_Instance(Excute := wire#w1, Aix_In := "输入轴驱动伺服", Parameter := "Modbus_Data".功能试验参数, Dir := False, Torque_In := "Modbus_Data_Rapid".传感器标定值[4], Stop := "程序停止", Done => #Temp[3], Busy =>, Error =>)
      Contact( #Temp[3] )
      Move(in := 123, out1 => "Modbus_Data_Rapid".设备状态)
   END_RUNG
   RUNG wire#powerrail
      { S7_Templates := "SrcType := Int" } EQ_Contact(in1 := "Modbus_Data_Rapid".设备状态, in2 := 122)
   END_RUNG wire#w1
   // the same network as SCL:
   #功能_Instance(Aix_In := "输入轴驱动伺服",   // "功能"
                Parameter := "Modbus_Data".功能试验参数,
                Excute := "Modbus_Data_Rapid".设备状态 = 122,
                Dir := False,
                Torque_In := "Modbus_Data_Rapid".传感器标定值[4],
                Stop := "程序停止",
                Done => #Temp[3],
                ENO => #_w1);
   IF #_w1 AND #Temp[3] THEN "Modbus_Data_Rapid".设备状态 := 123; END_IF;
END_REGION

REGION Network 9
   RUNG wire#powerrail
      #功能_Instance_1(Excute := wire#w1, Aix_In := "输入轴驱动伺服", Parameter := "Modbus_Data".功能试验参数, Dir := True, Torque_In := "Modbus_Data_Rapid".传感器标定值[4], Stop := "程序停止", Done => #Temp[4], Busy =>, Error =>)
      Contact( #Temp[4] )
      Move(in := 125, out1 => "Modbus_Data_Rapid".设备状态)
      R_Coil( "点火" )
   END_RUNG
   RUNG wire#powerrail
      { S7_Templates := "SrcType := Int" } EQ_Contact(in1 := "Modbus_Data_Rapid".设备状态, in2 := 124)
   END_RUNG wire#w1
   // the same network as SCL:
   #功能_Instance_1(Aix_In := "输入轴驱动伺服",   // "功能"
                  Parameter := "Modbus_Data".功能试验参数,
                  Excute := "Modbus_Data_Rapid".设备状态 = 124,
                  Dir := True,
                  Torque_In := "Modbus_Data_Rapid".传感器标定值[4],
                  Stop := "程序停止",
                  Done => #Temp[4],
                  ENO => #_w1);
   IF #_w1 AND #Temp[4] THEN
       "Modbus_Data_Rapid".设备状态 := 125;
       "点火" := FALSE;
   END_IF;
END_REGION

REGION Network 10
   RUNG wire#powerrail
      #力特性_Instance(Excute := wire#w1, Aix_In := "输入轴驱动伺服", Parameter := "Modbus_Data".力特性试验参数, Status := -2, Torque_In := "Modbus_Data_Rapid".传感器标定值[4], Stop := "程序停止", Done => #Temp[5], Busy =>, Error =>)
      Contact( #Temp[5] )
      Move(in := 131, out1 => "Modbus_Data_Rapid".设备状态)
   END_RUNG
   RUNG wire#powerrail
      { S7_Templates := "SrcType := Int" } EQ_Contact(in1 := "Modbus_Data_Rapid".设备状态, in2 := 130)
   END_RUNG wire#w1
   // the same network as SCL:
   #力特性_Instance(Aix_In := "输入轴驱动伺服",   // "力特性"
                 Parameter := "Modbus_Data".力特性试验参数,
                 Excute := "Modbus_Data_Rapid".设备状态 = 130,
                 Status := -2,
                 Torque_In := "Modbus_Data_Rapid".传感器标定值[4],
                 Stop := "程序停止",
                 Done => #Temp[5],
                 ENO => #_w1);
   IF #_w1 AND #Temp[5] THEN "Modbus_Data_Rapid".设备状态 := 131; END_IF;
END_REGION

REGION Network 11
   RUNG wire#powerrail
      #力特性_Instance_1(Excute := wire#w1, Aix_In := "输入轴驱动伺服", Parameter := "Modbus_Data".力特性试验参数, Status := -1, Torque_In := "Modbus_Data_Rapid".传感器标定值[4], Stop := "程序停止", Done => #Temp[6], Busy =>, Error =>)
      Contact( #Temp[6] )
      Move(in := 132, out1 => "Modbus_Data_Rapid".设备状态)
   END_RUNG
   RUNG wire#powerrail
      { S7_Templates := "SrcType := Int" } EQ_Contact(in1 := "Modbus_Data_Rapid".设备状态, in2 := 131)
   END_RUNG wire#w1
   // the same network as SCL:
   #力特性_Instance_1(Aix_In := "输入轴驱动伺服",   // "力特性"
                   Parameter := "Modbus_Data".力特性试验参数,
                   Excute := "Modbus_Data_Rapid".设备状态 = 131,
                   Status := -1,
                   Torque_In := "Modbus_Data_Rapid".传感器标定值[4],
                   Stop := "程序停止",
                   Done => #Temp[6],
                   ENO => #_w1);
   IF #_w1 AND #Temp[6] THEN "Modbus_Data_Rapid".设备状态 := 132; END_IF;
END_REGION

REGION Network 12
